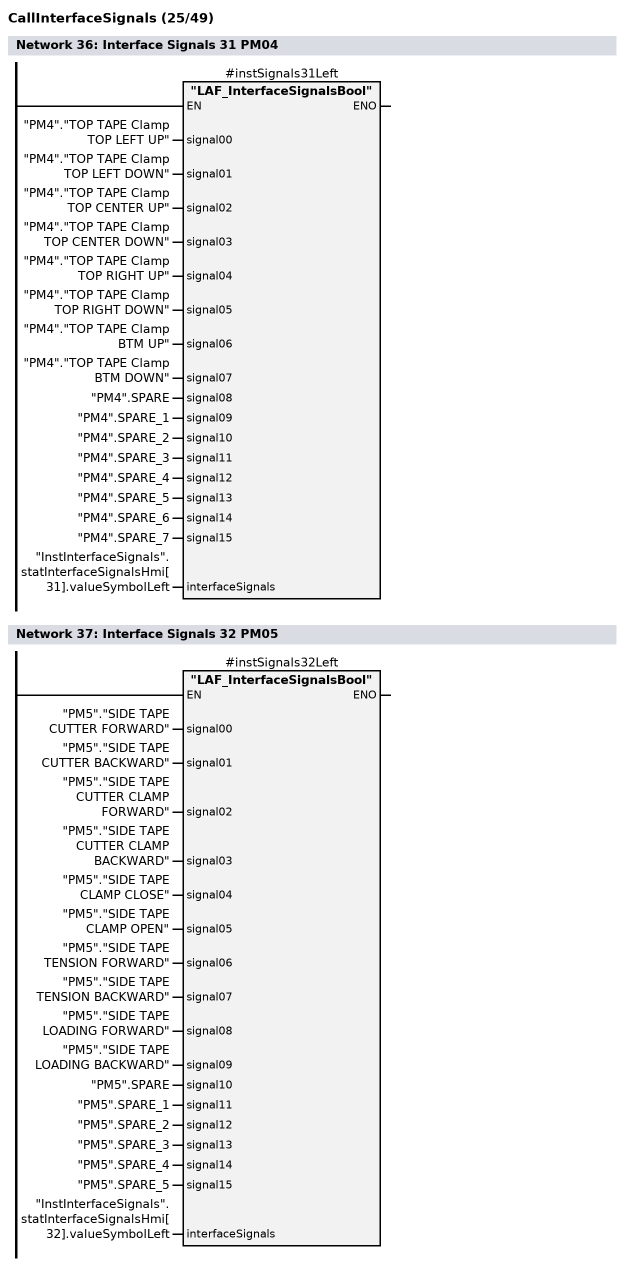
   RUNG wire#powerrail
      #instSignals31Left(signal00 := "PM4"."TOP TAPE Clamp TOP LEFT UP", signal01 := "PM4"."TOP TAPE Clamp TOP LEFT DOWN", signal02 := "PM4"."TOP TAPE Clamp TOP CENTER UP", signal03 := "PM4"."TOP TAPE Clamp TOP CENTER DOWN", signal04 := "PM4"."TOP TAPE Clamp TOP RIGHT UP", signal05 := "PM4"."TOP TAPE Clamp TOP RIGHT DOWN", signal06 := "PM4"."TOP TAPE Clamp BTM UP", signal07 := "PM4"."TOP TAPE Clamp BTM DOWN", signal08 := "PM4".SPARE, signal09 := "PM4".SPARE_1, signal10 := "PM4".SPARE_2, signal11 := "PM4".SPARE_3, signal12 := "PM4".SPARE_4, signal13 := "PM4".SPARE_5, signal14 := "PM4".SPARE_6, signal15 := "PM4".SPARE_7, interfaceSignals := "InstInterfaceSignals".statInterfaceSignalsHmi[31].valueSymbolLeft)
   END_RUNG
   // the same network as SCL:
   #instSignals31Left(signal00 := "PM4"."TOP TAPE Clamp TOP LEFT UP",   // "LAF_InterfaceSignalsBool"
                      signal01 := "PM4"."TOP TAPE Clamp TOP LEFT DOWN",
                      signal02 := "PM4"."TOP TAPE Clamp TOP CENTER UP",
                      signal03 := "PM4"."TOP TAPE Clamp TOP CENTER DOWN",
                      signal04 := "PM4"."TOP TAPE Clamp TOP RIGHT UP",
                      signal05 := "PM4"."TOP TAPE Clamp TOP RIGHT DOWN",
                      signal06 := "PM4"."TOP TAPE Clamp BTM UP",
                      signal07 := "PM4"."TOP TAPE Clamp BTM DOWN",
                      signal08 := "PM4".SPARE,
                      signal09 := "PM4".SPARE_1,
                      signal10 := "PM4".SPARE_2,
                      signal11 := "PM4".SPARE_3,
                      signal12 := "PM4".SPARE_4,
                      signal13 := "PM4".SPARE_5,
                      signal14 := "PM4".SPARE_6,
                      signal15 := "PM4".SPARE_7,
                      interfaceSignals := "InstInterfaceSignals".statInterfaceSignalsHmi[31].valueSymbolLeft);
END_REGION

REGION Network 37: Interface Signals 32 PM05
   RUNG wire#powerrail
      #instSignals32Left(signal00 := "PM5"."SIDE TAPE CUTTER FORWARD", signal01 := "PM5"."SIDE TAPE CUTTER BACKWARD", signal02 := "PM5"."SIDE TAPE CUTTER CLAMP FORWARD", signal03 := "PM5"."SIDE TAPE CUTTER CLAMP BACKWARD", signal04 := "PM5"."SIDE TAPE CLAMP CLOSE", signal05 := "PM5"."SIDE TAPE CLAMP OPEN", signal06 := "PM5"."SIDE TAPE TENSION FORWARD", signal07 := "PM5"."SIDE TAPE TENSION BACKWARD", signal08 := "PM5"."SIDE TAPE LOADING FORWARD", signal09 := "PM5"."SIDE TAPE LOADING BACKWARD", signal10 := "PM5".SPARE, signal11 := "PM5".SPARE_1, signal12 := "PM5".SPARE_2, signal13 := "PM5".SPARE_3, signal14 := "PM5".SPARE_4, signal15 := "PM5".SPARE_5, interfaceSignals := "InstInterfaceSignals".statInterfaceSignalsHmi[32].valueSymbolLeft)
   END_RUNG
   // the same network as SCL:
   #instSignals32Left(signal00 := "PM5"."SIDE TAPE CUTTER FORWARD",   // "LAF_InterfaceSignalsBool"
                      signal01 := "PM5"."SIDE TAPE CUTTER BACKWARD",
                      signal02 := "PM5"."SIDE TAPE CUTTER CLAMP FORWARD",
                      signal03 := "PM5"."SIDE TAPE CUTTER CLAMP BACKWARD",
                      signal04 := "PM5"."SIDE TAPE CLAMP CLOSE",
                      signal05 := "PM5"."SIDE TAPE CLAMP OPEN",
                      signal06 := "PM5"."SIDE TAPE TENSION FORWARD",
                      signal07 := "PM5"."SIDE TAPE TENSION BACKWARD",
                      signal08 := "PM5"."SIDE TAPE LOADING FORWARD",
                      signal09 := "PM5"."SIDE TAPE LOADING BACKWARD",
                      signal10 := "PM5".SPARE,
                      signal11 := "PM5".SPARE_1,
                      signal12 := "PM5".SPARE_2,
                      signal13 := "PM5".SPARE_3,
                      signal14 := "PM5".SPARE_4,
                      signal15 := "PM5".SPARE_5,
                      interfaceSignals := "InstInterfaceSignals".statInterfaceSignalsHmi[32].valueSymbolLeft);
END_REGION

REGION Network 38: Interface Signals 33 PM06
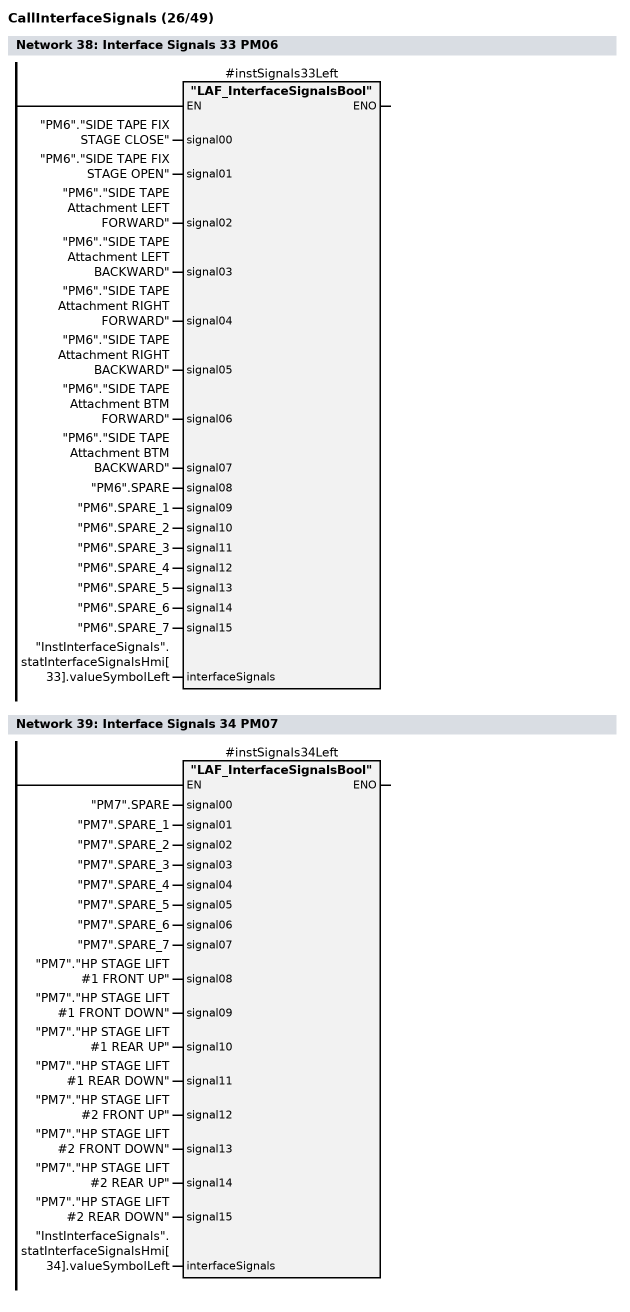
   RUNG wire#powerrail
      #instSignals33Left(signal00 := "PM6"."SIDE TAPE FIX STAGE CLOSE", signal01 := "PM6"."SIDE TAPE FIX STAGE OPEN", signal02 := "PM6"."SIDE TAPE Attachment LEFT FORWARD", signal03 := "PM6"."SIDE TAPE Attachment LEFT BACKWARD", signal04 := "PM6"."SIDE TAPE Attachment RIGHT FORWARD", signal05 := "PM6"."SIDE TAPE Attachment RIGHT BACKWARD", signal06 := "PM6"."SIDE TAPE Attachment BTM FORWARD", signal07 := "PM6"."SIDE TAPE Attachment BTM BACKWARD", signal08 := "PM6".SPARE, signal09 := "PM6".SPARE_1, signal10 := "PM6".SPARE_2, signal11 := "PM6".SPARE_3, signal12 := "PM6".SPARE_4, signal13 := "PM6".SPARE_5, signal14 := "PM6".SPARE_6, signal15 := "PM6".SPARE_7, interfaceSignals := "InstInterfaceSignals".statInterfaceSignalsHmi[33].valueSymbolLeft)
   END_RUNG
   // the same network as SCL:
   #instSignals33Left(signal00 := "PM6"."SIDE TAPE FIX STAGE CLOSE",   // "LAF_InterfaceSignalsBool"
                      signal01 := "PM6"."SIDE TAPE FIX STAGE OPEN",
                      signal02 := "PM6"."SIDE TAPE Attachment LEFT FORWARD",
                      signal03 := "PM6"."SIDE TAPE Attachment LEFT BACKWARD",
                      signal04 := "PM6"."SIDE TAPE Attachment RIGHT FORWARD",
                      signal05 := "PM6"."SIDE TAPE Attachment RIGHT BACKWARD",
                      signal06 := "PM6"."SIDE TAPE Attachment BTM FORWARD",
                      signal07 := "PM6"."SIDE TAPE Attachment BTM BACKWARD",
                      signal08 := "PM6".SPARE,
                      signal09 := "PM6".SPARE_1,
                      signal10 := "PM6".SPARE_2,
                      signal11 := "PM6".SPARE_3,
                      signal12 := "PM6".SPARE_4,
                      signal13 := "PM6".SPARE_5,
                      signal14 := "PM6".SPARE_6,
                      signal15 := "PM6".SPARE_7,
                      interfaceSignals := "InstInterfaceSignals".statInterfaceSignalsHmi[33].valueSymbolLeft);
END_REGION

REGION Network 39: Interface Signals 34 PM07
   RUNG wire#powerrail
      #instSignals34Left(signal00 := "PM7".SPARE, signal01 := "PM7".SPARE_1, signal02 := "PM7".SPARE_2, signal03 := "PM7".SPARE_3, signal04 := "PM7".SPARE_4, signal05 := "PM7".SPARE_5, signal06 := "PM7".SPARE_6, signal07 := "PM7".SPARE_7, signal08 := "PM7"."HP STAGE LIFT #1 FRONT UP", signal09 := "PM7"."HP STAGE LIFT #1 FRONT DOWN", signal10 := "PM7"."HP STAGE LIFT #1 REAR UP", signal11 := "PM7"."HP STAGE LIFT #1 REAR DOWN", signal12 := "PM7"."HP STAGE LIFT #2 FRONT UP", signal13 := "PM7"."HP STAGE LIFT #2 FRONT DOWN", signal14 := "PM7"."HP STAGE LIFT #2 REAR UP", signal15 := "PM7"."HP STAGE LIFT #2 REAR DOWN", interfaceSignals := "InstInterfaceSignals".statInterfaceSignalsHmi[34].valueSymbolLeft)
   END_RUNG
   // the same network as SCL:
   #instSignals34Left(signal00 := "PM7".SPARE,   // "LAF_InterfaceSignalsBool"
                      signal01 := "PM7".SPARE_1,
                      signal02 := "PM7".SPARE_2,
                      signal03 := "PM7".SPARE_3,
                      signal04 := "PM7".SPARE_4,
                      signal05 := "PM7".SPARE_5,
                      signal06 := "PM7".SPARE_6,
                      signal07 := "PM7".SPARE_7,
                      signal08 := "PM7"."HP STAGE LIFT #1 FRONT UP",
                      signal09 := "PM7"."HP STAGE LIFT #1 FRONT DOWN",
                      signal10 := "PM7"."HP STAGE LIFT #1 REAR UP",
                      signal11 := "PM7"."HP STAGE LIFT #1 REAR DOWN",
                      signal12 := "PM7"."HP STAGE LIFT #2 FRONT UP",
                      signal13 := "PM7"."HP STAGE LIFT #2 FRONT DOWN",
                      signal14 := "PM7"."HP STAGE LIFT #2 REAR UP",
                      signal15 := "PM7"."HP STAGE LIFT #2 REAR DOWN",
                      interfaceSignals := "InstInterfaceSignals".statInterfaceSignalsHmi[34].valueSymbolLeft);
END_REGION

REGION Network 40: Interface Signals 35 PM08
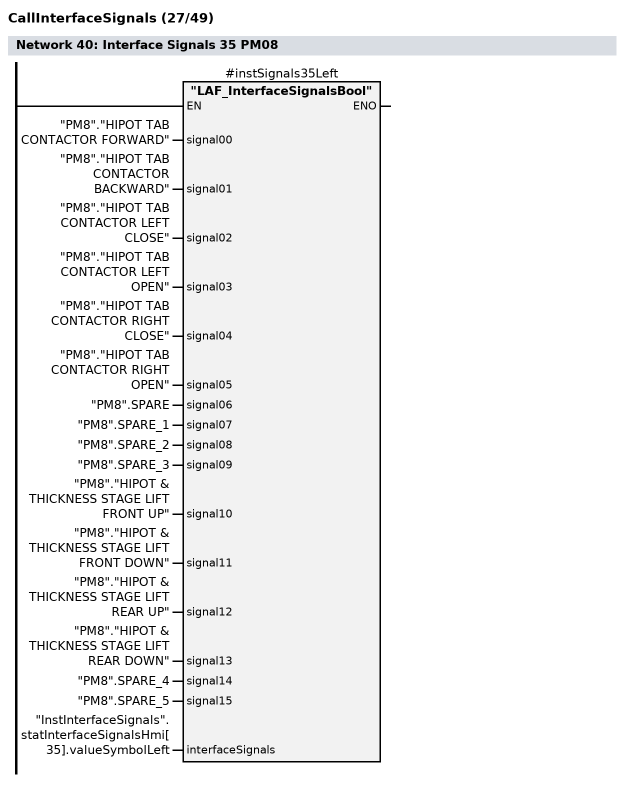
   RUNG wire#powerrail
      #instSignals35Left(signal00 := "PM8"."HIPOT TAB CONTACTOR FORWARD", signal01 := "PM8"."HIPOT TAB CONTACTOR BACKWARD", signal02 := "PM8"."HIPOT TAB CONTACTOR LEFT CLOSE", signal03 := "PM8"."HIPOT TAB CONTACTOR LEFT OPEN", signal04 := "PM8"."HIPOT TAB CONTACTOR RIGHT CLOSE", signal05 := "PM8"."HIPOT TAB CONTACTOR RIGHT OPEN", signal06 := "PM8".SPARE, signal07 := "PM8".SPARE_1, signal08 := "PM8".SPARE_2, signal09 := "PM8".SPARE_3, signal10 := "PM8"."HIPOT & THICKNESS STAGE LIFT FRONT UP", signal11 := "PM8"."HIPOT & THICKNESS STAGE LIFT FRONT DOWN", signal12 := "PM8"."HIPOT & THICKNESS STAGE LIFT REAR UP", signal13 := "PM8"."HIPOT & THICKNESS STAGE LIFT REAR DOWN", signal14 := "PM8".SPARE_4, signal15 := "PM8".SPARE_5, interfaceSignals := "InstInterfaceSignals".statInterfaceSignalsHmi[35].valueSymbolLeft)
   END_RUNG
   // the same network as SCL:
   #instSignals35Left(signal00 := "PM8"."HIPOT TAB CONTACTOR FORWARD",   // "LAF_InterfaceSignalsBool"
                      signal01 := "PM8"."HIPOT TAB CONTACTOR BACKWARD",
                      signal02 := "PM8"."HIPOT TAB CONTACTOR LEFT CLOSE",
                      signal03 := "PM8"."HIPOT TAB CONTACTOR LEFT OPEN",
                      signal04 := "PM8"."HIPOT TAB CONTACTOR RIGHT CLOSE",
                      signal05 := "PM8"."HIPOT TAB CONTACTOR RIGHT OPEN",
                      signal06 := "PM8".SPARE,
                      signal07 := "PM8".SPARE_1,
                      signal08 := "PM8".SPARE_2,
                      signal09 := "PM8".SPARE_3,
                      signal10 := "PM8"."HIPOT & THICKNESS STAGE LIFT FRONT UP",
                      signal11 := "PM8"."HIPOT & THICKNESS STAGE LIFT FRONT DOWN",
                      signal12 := "PM8"."HIPOT & THICKNESS STAGE LIFT REAR UP",
                      signal13 := "PM8"."HIPOT & THICKNESS STAGE LIFT REAR DOWN",
                      signal14 := "PM8".SPARE_4,
                      signal15 := "PM8".SPARE_5,
                      interfaceSignals := "InstInterfaceSignals".statInterfaceSignalsHmi[35].valueSymbolLeft);
END_REGION

REGION Network 41: Interface Signals 36 PM09
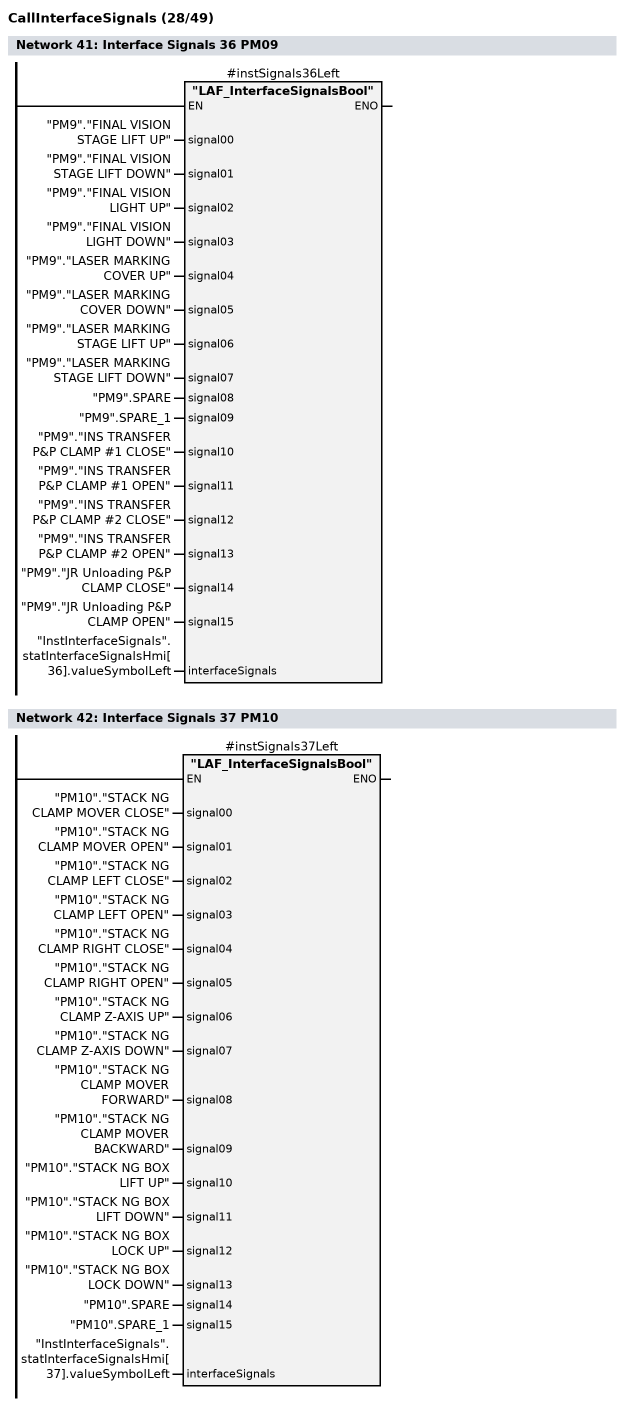
   RUNG wire#powerrail
      #instSignals36Left(signal00 := "PM9"."FINAL VISION STAGE LIFT UP", signal01 := "PM9"."FINAL VISION STAGE LIFT DOWN", signal02 := "PM9"."FINAL VISION LIGHT UP", signal03 := "PM9"."FINAL VISION LIGHT DOWN", signal04 := "PM9"."LASER MARKING COVER UP", signal05 := "PM9"."LASER MARKING COVER DOWN", signal06 := "PM9"."LASER MARKING STAGE LIFT UP", signal07 := "PM9"."LASER MARKING STAGE LIFT DOWN", signal08 := "PM9".SPARE, signal09 := "PM9".SPARE_1, signal10 := "PM9"."INS TRANSFER P&P CLAMP #1 CLOSE", signal11 := "PM9"."INS TRANSFER P&P CLAMP #1 OPEN", signal12 := "PM9"."INS TRANSFER P&P CLAMP #2 CLOSE", signal13 := "PM9"."INS TRANSFER P&P CLAMP #2 OPEN", signal14 := "PM9"."JR Unloading P&P CLAMP CLOSE", signal15 := "PM9"."JR Unloading P&P CLAMP OPEN", interfaceSignals := "InstInterfaceSignals".statInterfaceSignalsHmi[36].valueSymbolLeft)
   END_RUNG
   // the same network as SCL:
   #instSignals36Left(signal00 := "PM9"."FINAL VISION STAGE LIFT UP",   // "LAF_InterfaceSignalsBool"
                      signal01 := "PM9"."FINAL VISION STAGE LIFT DOWN",
                      signal02 := "PM9"."FINAL VISION LIGHT UP",
                      signal03 := "PM9"."FINAL VISION LIGHT DOWN",
                      signal04 := "PM9"."LASER MARKING COVER UP",
                      signal05 := "PM9"."LASER MARKING COVER DOWN",
                      signal06 := "PM9"."LASER MARKING STAGE LIFT UP",
                      signal07 := "PM9"."LASER MARKING STAGE LIFT DOWN",
                      signal08 := "PM9".SPARE,
                      signal09 := "PM9".SPARE_1,
                      signal10 := "PM9"."INS TRANSFER P&P CLAMP #1 CLOSE",
                      signal11 := "PM9"."INS TRANSFER P&P CLAMP #1 OPEN",
                      signal12 := "PM9"."INS TRANSFER P&P CLAMP #2 CLOSE",
                      signal13 := "PM9"."INS TRANSFER P&P CLAMP #2 OPEN",
                      signal14 := "PM9"."JR Unloading P&P CLAMP CLOSE",
                      signal15 := "PM9"."JR Unloading P&P CLAMP OPEN",
                      interfaceSignals := "InstInterfaceSignals".statInterfaceSignalsHmi[36].valueSymbolLeft);
END_REGION

REGION Network 42: Interface Signals 37 PM10
   RUNG wire#powerrail
      #instSignals37Left(signal00 := "PM10"."STACK NG CLAMP MOVER CLOSE", signal01 := "PM10"."STACK NG CLAMP MOVER OPEN", signal02 := "PM10"."STACK NG CLAMP LEFT CLOSE", signal03 := "PM10"."STACK NG CLAMP LEFT OPEN", signal04 := "PM10"."STACK NG CLAMP RIGHT CLOSE", signal05 := "PM10"."STACK NG CLAMP RIGHT OPEN", signal06 := "PM10"."STACK NG CLAMP Z-AXIS UP", signal07 := "PM10"."STACK NG CLAMP Z-AXIS DOWN", signal08 := "PM10"."STACK NG CLAMP MOVER FORWARD", signal09 := "PM10"."STACK NG CLAMP MOVER BACKWARD", signal10 := "PM10"."STACK NG BOX LIFT UP", signal11 := "PM10"."STACK NG BOX LIFT DOWN", signal12 := "PM10"."STACK NG BOX LOCK UP", signal13 := "PM10"."STACK NG BOX LOCK DOWN", signal14 := "PM10".SPARE, signal15 := "PM10".SPARE_1, interfaceSignals := "InstInterfaceSignals".statInterfaceSignalsHmi[37].valueSymbolLeft)
   END_RUNG
   // the same network as SCL:
   #instSignals37Left(signal00 := "PM10"."STACK NG CLAMP MOVER CLOSE",   // "LAF_InterfaceSignalsBool"
                      signal01 := "PM10"."STACK NG CLAMP MOVER OPEN",
                      signal02 := "PM10"."STACK NG CLAMP LEFT CLOSE",
                      signal03 := "PM10"."STACK NG CLAMP LEFT OPEN",
                      signal04 := "PM10"."STACK NG CLAMP RIGHT CLOSE",
                      signal05 := "PM10"."STACK NG CLAMP RIGHT OPEN",
                      signal06 := "PM10"."STACK NG CLAMP Z-AXIS UP",
                      signal07 := "PM10"."STACK NG CLAMP Z-AXIS DOWN",
                      signal08 := "PM10"."STACK NG CLAMP MOVER FORWARD",
                      signal09 := "PM10"."STACK NG CLAMP MOVER BACKWARD",
                      signal10 := "PM10"."STACK NG BOX LIFT UP",
                      signal11 := "PM10"."STACK NG BOX LIFT DOWN",
                      signal12 := "PM10"."STACK NG BOX LOCK UP",
                      signal13 := "PM10"."STACK NG BOX LOCK DOWN",
                      signal14 := "PM10".SPARE,
                      signal15 := "PM10".SPARE_1,
                      interfaceSignals := "InstInterfaceSignals".statInterfaceSignalsHmi[37].valueSymbolLeft);
END_REGION

REGION Network 43: Interface Signals 38 SBK01
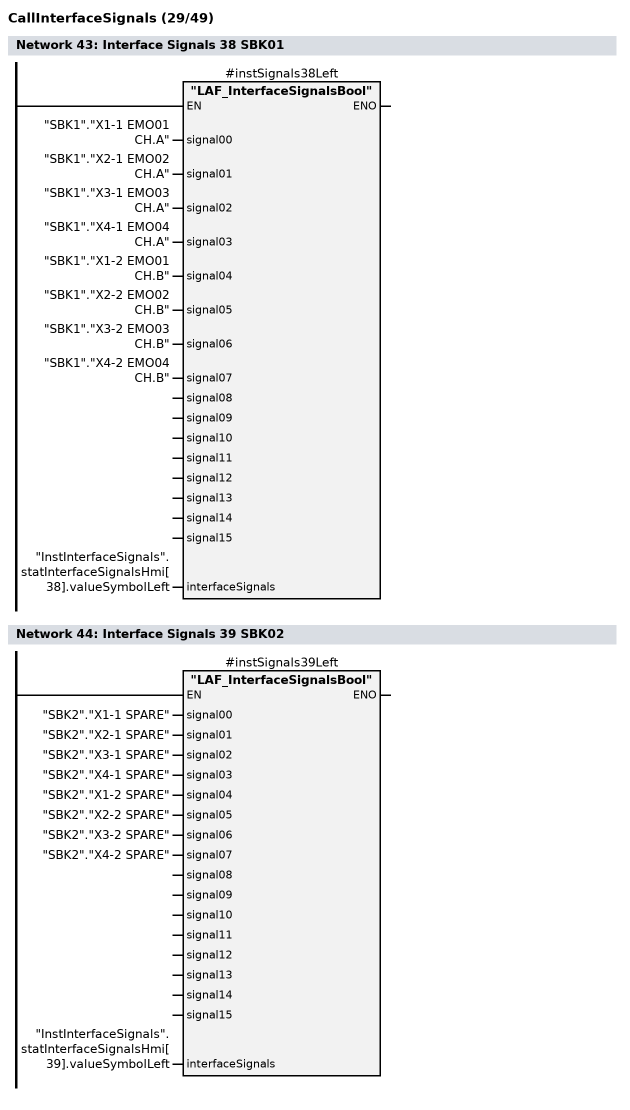
   RUNG wire#powerrail
      #instSignals38Left(signal00 := "SBK1"."X1-1 EMO01 CH.A", signal01 := "SBK1"."X2-1 EMO02 CH.A", signal02 := "SBK1"."X3-1 EMO03 CH.A", signal03 := "SBK1"."X4-1 EMO04 CH.A", signal04 := "SBK1"."X1-2 EMO01 CH.B", signal05 := "SBK1"."X2-2 EMO02 CH.B", signal06 := "SBK1"."X3-2 EMO03 CH.B", signal07 := "SBK1"."X4-2 EMO04 CH.B", signal08 :=, signal09 :=, signal10 :=, signal11 :=, signal12 :=, signal13 :=, signal14 :=, signal15 :=, interfaceSignals := "InstInterfaceSignals".statInterfaceSignalsHmi[38].valueSymbolLeft)
   END_RUNG
   // the same network as SCL:
   #instSignals38Left(signal00 := "SBK1"."X1-1 EMO01 CH.A",   // "LAF_InterfaceSignalsBool"
                      signal01 := "SBK1"."X2-1 EMO02 CH.A",
                      signal02 := "SBK1"."X3-1 EMO03 CH.A",
                      signal03 := "SBK1"."X4-1 EMO04 CH.A",
                      signal04 := "SBK1"."X1-2 EMO01 CH.B",
                      signal05 := "SBK1"."X2-2 EMO02 CH.B",
                      signal06 := "SBK1"."X3-2 EMO03 CH.B",
                      signal07 := "SBK1"."X4-2 EMO04 CH.B",
                      interfaceSignals := "InstInterfaceSignals".statInterfaceSignalsHmi[38].valueSymbolLeft);
END_REGION

REGION Network 44: Interface Signals 39 SBK02
   RUNG wire#powerrail
      #instSignals39Left(signal00 := "SBK2"."X1-1 SPARE", signal01 := "SBK2"."X2-1 SPARE", signal02 := "SBK2"."X3-1 SPARE", signal03 := "SBK2"."X4-1 SPARE", signal04 := "SBK2"."X1-2 SPARE", signal05 := "SBK2"."X2-2 SPARE", signal06 := "SBK2"."X3-2 SPARE", signal07 := "SBK2"."X4-2 SPARE", signal08 :=, signal09 :=, signal10 :=, signal11 :=, signal12 :=, signal13 :=, signal14 :=, signal15 :=, interfaceSignals := "InstInterfaceSignals".statInterfaceSignalsHmi[39].valueSymbolLeft)
   END_RUNG
   // the same network as SCL:
   #instSignals39Left(signal00 := "SBK2"."X1-1 SPARE",   // "LAF_InterfaceSignalsBool"
                      signal01 := "SBK2"."X2-1 SPARE",
                      signal02 := "SBK2"."X3-1 SPARE",
                      signal03 := "SBK2"."X4-1 SPARE",
                      signal04 := "SBK2"."X1-2 SPARE",
                      signal05 := "SBK2"."X2-2 SPARE",
                      signal06 := "SBK2"."X3-2 SPARE",
                      signal07 := "SBK2"."X4-2 SPARE",
                      interfaceSignals := "InstInterfaceSignals".statInterfaceSignalsHmi[39].valueSymbolLeft);
END_REGION

REGION Network 45: Interface Signals 40 SBK03
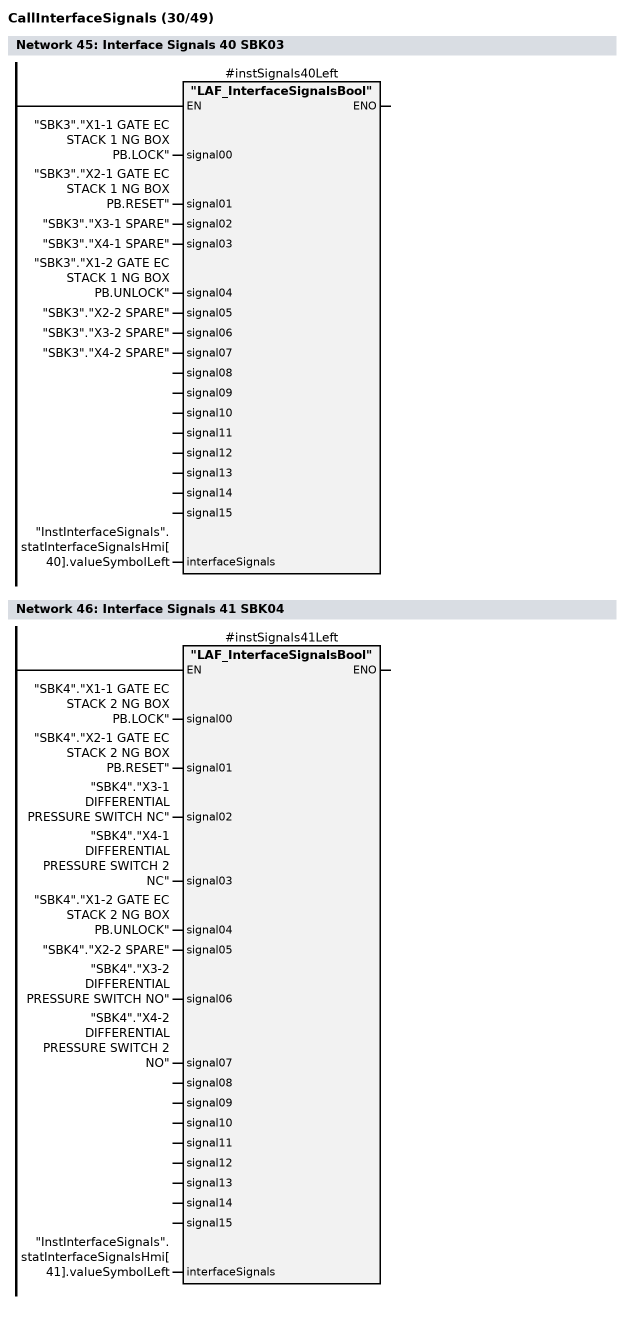
   RUNG wire#powerrail
      #instSignals40Left(signal00 := "SBK3"."X1-1 GATE EC STACK 1 NG BOX PB.LOCK", signal01 := "SBK3"."X2-1 GATE EC STACK 1 NG BOX PB.RESET", signal02 := "SBK3"."X3-1 SPARE", signal03 := "SBK3"."X4-1 SPARE", signal04 := "SBK3"."X1-2 GATE EC STACK 1 NG BOX PB.UNLOCK", signal05 := "SBK3"."X2-2 SPARE", signal06 := "SBK3"."X3-2 SPARE", signal07 := "SBK3"."X4-2 SPARE", signal08 :=, signal09 :=, signal10 :=, signal11 :=, signal12 :=, signal13 :=, signal14 :=, signal15 :=, interfaceSignals := "InstInterfaceSignals".statInterfaceSignalsHmi[40].valueSymbolLeft)
   END_RUNG
   // the same network as SCL:
   #instSignals40Left(signal00 := "SBK3"."X1-1 GATE EC STACK 1 NG BOX PB.LOCK",   // "LAF_InterfaceSignalsBool"
                      signal01 := "SBK3"."X2-1 GATE EC STACK 1 NG BOX PB.RESET",
                      signal02 := "SBK3"."X3-1 SPARE",
                      signal03 := "SBK3"."X4-1 SPARE",
                      signal04 := "SBK3"."X1-2 GATE EC STACK 1 NG BOX PB.UNLOCK",
                      signal05 := "SBK3"."X2-2 SPARE",
                      signal06 := "SBK3"."X3-2 SPARE",
                      signal07 := "SBK3"."X4-2 SPARE",
                      interfaceSignals := "InstInterfaceSignals".statInterfaceSignalsHmi[40].valueSymbolLeft);
END_REGION

REGION Network 46: Interface Signals 41 SBK04
   RUNG wire#powerrail
      #instSignals41Left(signal00 := "SBK4"."X1-1 GATE EC STACK 2 NG BOX PB.LOCK", signal01 := "SBK4"."X2-1 GATE EC STACK 2 NG BOX PB.RESET", signal02 := "SBK4"."X3-1 DIFFERENTIAL PRESSURE SWITCH NC", signal03 := "SBK4"."X4-1 DIFFERENTIAL PRESSURE SWITCH 2 NC", signal04 := "SBK4"."X1-2 GATE EC STACK 2 NG BOX PB.UNLOCK", signal05 := "SBK4"."X2-2 SPARE", signal06 := "SBK4"."X3-2 DIFFERENTIAL PRESSURE SWITCH NO", signal07 := "SBK4"."X4-2 DIFFERENTIAL PRESSURE SWITCH 2 NO", signal08 :=, signal09 :=, signal10 :=, signal11 :=, signal12 :=, signal13 :=, signal14 :=, signal15 :=, interfaceSignals := "InstInterfaceSignals".statInterfaceSignalsHmi[41].valueSymbolLeft)
   END_RUNG
   // the same network as SCL:
   #instSignals41Left(signal00 := "SBK4"."X1-1 GATE EC STACK 2 NG BOX PB.LOCK",   // "LAF_InterfaceSignalsBool"
                      signal01 := "SBK4"."X2-1 GATE EC STACK 2 NG BOX PB.RESET",
                      signal02 := "SBK4"."X3-1 DIFFERENTIAL PRESSURE SWITCH NC",
                      signal03 := "SBK4"."X4-1 DIFFERENTIAL PRESSURE SWITCH 2 NC",
                      signal04 := "SBK4"."X1-2 GATE EC STACK 2 NG BOX PB.UNLOCK",
                      signal05 := "SBK4"."X2-2 SPARE",
                      signal06 := "SBK4"."X3-2 DIFFERENTIAL PRESSURE SWITCH NO",
                      signal07 := "SBK4"."X4-2 DIFFERENTIAL PRESSURE SWITCH 2 NO",
                      interfaceSignals := "InstInterfaceSignals".statInterfaceSignalsHmi[41].valueSymbolLeft);
END_REGION

REGION Network 47: Interface Signals 42 SBK05
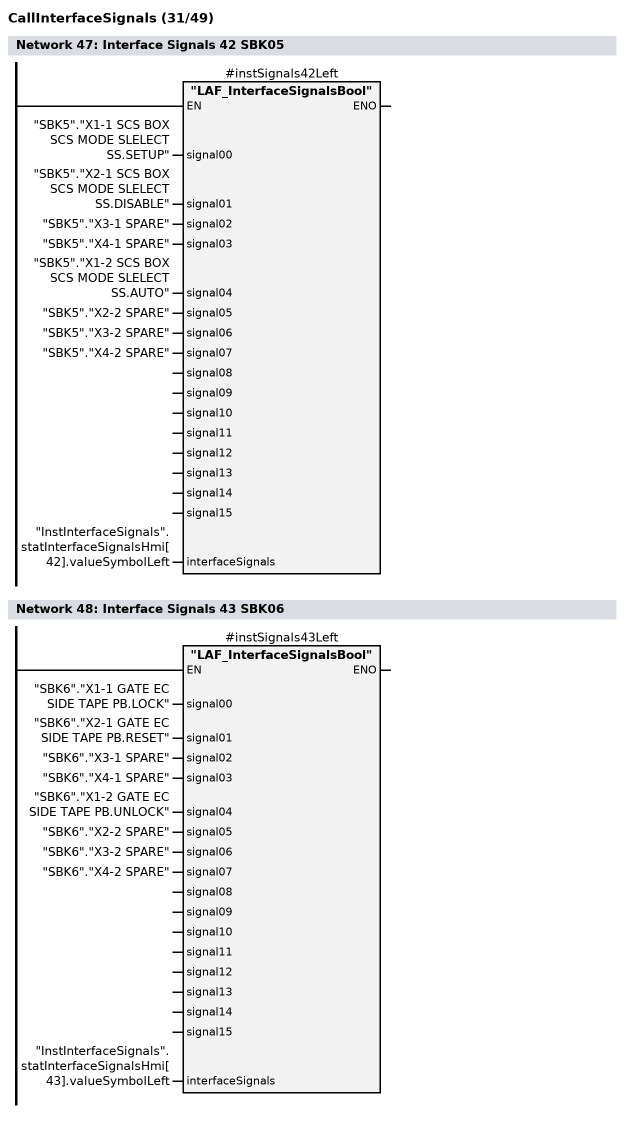
   RUNG wire#powerrail
      #instSignals42Left(signal00 := "SBK5"."X1-1 SCS BOX SCS MODE SLELECT SS.SETUP", signal01 := "SBK5"."X2-1 SCS BOX SCS MODE SLELECT SS.DISABLE", signal02 := "SBK5"."X3-1 SPARE", signal03 := "SBK5"."X4-1 SPARE", signal04 := "SBK5"."X1-2 SCS BOX SCS MODE SLELECT SS.AUTO", signal05 := "SBK5"."X2-2 SPARE", signal06 := "SBK5"."X3-2 SPARE", signal07 := "SBK5"."X4-2 SPARE", signal08 :=, signal09 :=, signal10 :=, signal11 :=, signal12 :=, signal13 :=, signal14 :=, signal15 :=, interfaceSignals := "InstInterfaceSignals".statInterfaceSignalsHmi[42].valueSymbolLeft)
   END_RUNG
   // the same network as SCL:
   #instSignals42Left(signal00 := "SBK5"."X1-1 SCS BOX SCS MODE SLELECT SS.SETUP",   // "LAF_InterfaceSignalsBool"
                      signal01 := "SBK5"."X2-1 SCS BOX SCS MODE SLELECT SS.DISABLE",
                      signal02 := "SBK5"."X3-1 SPARE",
                      signal03 := "SBK5"."X4-1 SPARE",
                      signal04 := "SBK5"."X1-2 SCS BOX SCS MODE SLELECT SS.AUTO",
                      signal05 := "SBK5"."X2-2 SPARE",
                      signal06 := "SBK5"."X3-2 SPARE",
                      signal07 := "SBK5"."X4-2 SPARE",
                      interfaceSignals := "InstInterfaceSignals".statInterfaceSignalsHmi[42].valueSymbolLeft);
END_REGION

REGION Network 48: Interface Signals 43 SBK06
   RUNG wire#powerrail
      #instSignals43Left(signal00 := "SBK6"."X1-1 GATE EC SIDE TAPE PB.LOCK", signal01 := "SBK6"."X2-1 GATE EC SIDE TAPE PB.RESET", signal02 := "SBK6"."X3-1 SPARE", signal03 := "SBK6"."X4-1 SPARE", signal04 := "SBK6"."X1-2 GATE EC SIDE TAPE PB.UNLOCK", signal05 := "SBK6"."X2-2 SPARE", signal06 := "SBK6"."X3-2 SPARE", signal07 := "SBK6"."X4-2 SPARE", signal08 :=, signal09 :=, signal10 :=, signal11 :=, signal12 :=, signal13 :=, signal14 :=, signal15 :=, interfaceSignals := "InstInterfaceSignals".statInterfaceSignalsHmi[43].valueSymbolLeft)
   END_RUNG
   // the same network as SCL:
   #instSignals43Left(signal00 := "SBK6"."X1-1 GATE EC SIDE TAPE PB.LOCK",   // "LAF_InterfaceSignalsBool"
                      signal01 := "SBK6"."X2-1 GATE EC SIDE TAPE PB.RESET",
                      signal02 := "SBK6"."X3-1 SPARE",
                      signal03 := "SBK6"."X4-1 SPARE",
                      signal04 := "SBK6"."X1-2 GATE EC SIDE TAPE PB.UNLOCK",
                      signal05 := "SBK6"."X2-2 SPARE",
                      signal06 := "SBK6"."X3-2 SPARE",
                      signal07 := "SBK6"."X4-2 SPARE",
                      interfaceSignals := "InstInterfaceSignals".statInterfaceSignalsHmi[43].valueSymbolLeft);
END_REGION

REGION Network 49: Interface Signals 44 SBK07
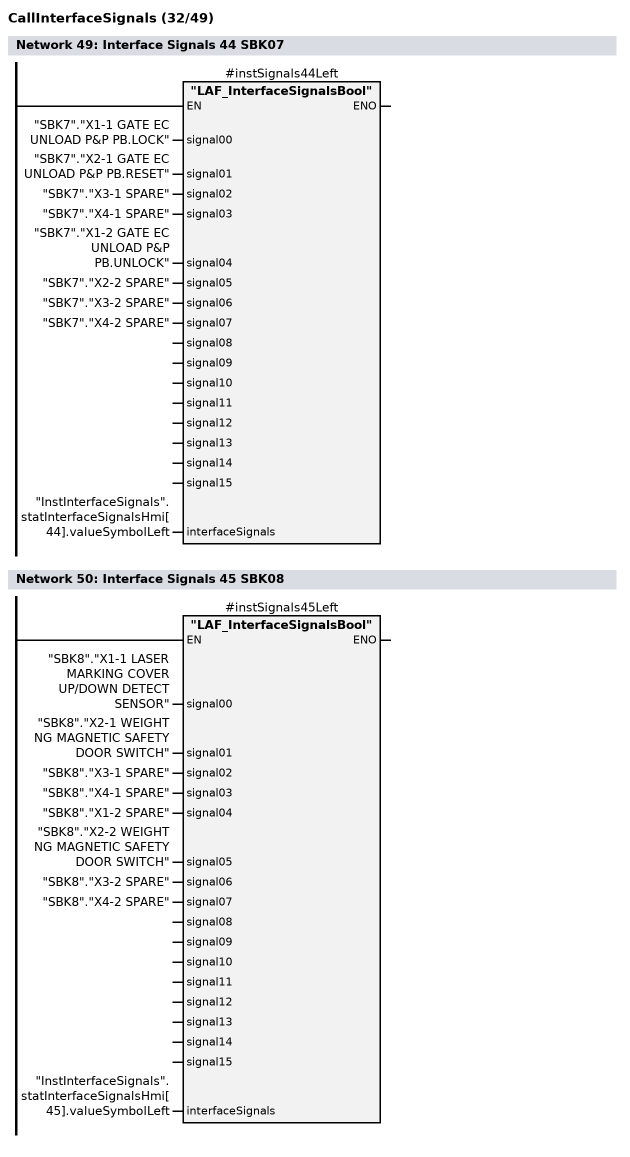
   RUNG wire#powerrail
      #instSignals44Left(signal00 := "SBK7"."X1-1 GATE EC UNLOAD P&P PB.LOCK", signal01 := "SBK7"."X2-1 GATE EC UNLOAD P&P PB.RESET", signal02 := "SBK7"."X3-1 SPARE", signal03 := "SBK7"."X4-1 SPARE", signal04 := "SBK7"."X1-2 GATE EC UNLOAD P&P PB.UNLOCK", signal05 := "SBK7"."X2-2 SPARE", signal06 := "SBK7"."X3-2 SPARE", signal07 := "SBK7"."X4-2 SPARE", signal08 :=, signal09 :=, signal10 :=, signal11 :=, signal12 :=, signal13 :=, signal14 :=, signal15 :=, interfaceSignals := "InstInterfaceSignals".statInterfaceSignalsHmi[44].valueSymbolLeft)
   END_RUNG
   // the same network as SCL:
   #instSignals44Left(signal00 := "SBK7"."X1-1 GATE EC UNLOAD P&P PB.LOCK",   // "LAF_InterfaceSignalsBool"
                      signal01 := "SBK7"."X2-1 GATE EC UNLOAD P&P PB.RESET",
                      signal02 := "SBK7"."X3-1 SPARE",
                      signal03 := "SBK7"."X4-1 SPARE",
                      signal04 := "SBK7"."X1-2 GATE EC UNLOAD P&P PB.UNLOCK",
                      signal05 := "SBK7"."X2-2 SPARE",
                      signal06 := "SBK7"."X3-2 SPARE",
                      signal07 := "SBK7"."X4-2 SPARE",
                      interfaceSignals := "InstInterfaceSignals".statInterfaceSignalsHmi[44].valueSymbolLeft);
END_REGION

REGION Network 50: Interface Signals 45 SBK08
   RUNG wire#powerrail
      #instSignals45Left(signal00 := "SBK8"."X1-1 LASER MARKING COVER UP/DOWN DETECT SENSOR", signal01 := "SBK8"."X2-1 WEIGHT NG MAGNETIC SAFETY DOOR SWITCH", signal02 := "SBK8"."X3-1 SPARE", signal03 := "SBK8"."X4-1 SPARE", signal04 := "SBK8"."X1-2 SPARE", signal05 := "SBK8"."X2-2 WEIGHT NG MAGNETIC SAFETY DOOR SWITCH", signal06 := "SBK8"."X3-2 SPARE", signal07 := "SBK8"."X4-2 SPARE", signal08 :=, signal09 :=, signal10 :=, signal11 :=, signal12 :=, signal13 :=, signal14 :=, signal15 :=, interfaceSignals := "InstInterfaceSignals".statInterfaceSignalsHmi[45].valueSymbolLeft)
   END_RUNG
   // the same network as SCL:
   #instSignals45Left(signal00 := "SBK8"."X1-1 LASER MARKING COVER UP/DOWN DETECT SENSOR",   // "LAF_InterfaceSignalsBool"
                      signal01 := "SBK8"."X2-1 WEIGHT NG MAGNETIC SAFETY DOOR SWITCH",
                      signal02 := "SBK8"."X3-1 SPARE",
                      signal03 := "SBK8"."X4-1 SPARE",
                      signal04 := "SBK8"."X1-2 SPARE",
                      signal05 := "SBK8"."X2-2 WEIGHT NG MAGNETIC SAFETY DOOR SWITCH",
                      signal06 := "SBK8"."X3-2 SPARE",
                      signal07 := "SBK8"."X4-2 SPARE",
                      interfaceSignals := "InstInterfaceSignals".statInterfaceSignalsHmi[45].valueSymbolLeft);
END_REGION

REGION Network 51: Interface Signals 46 SBK09
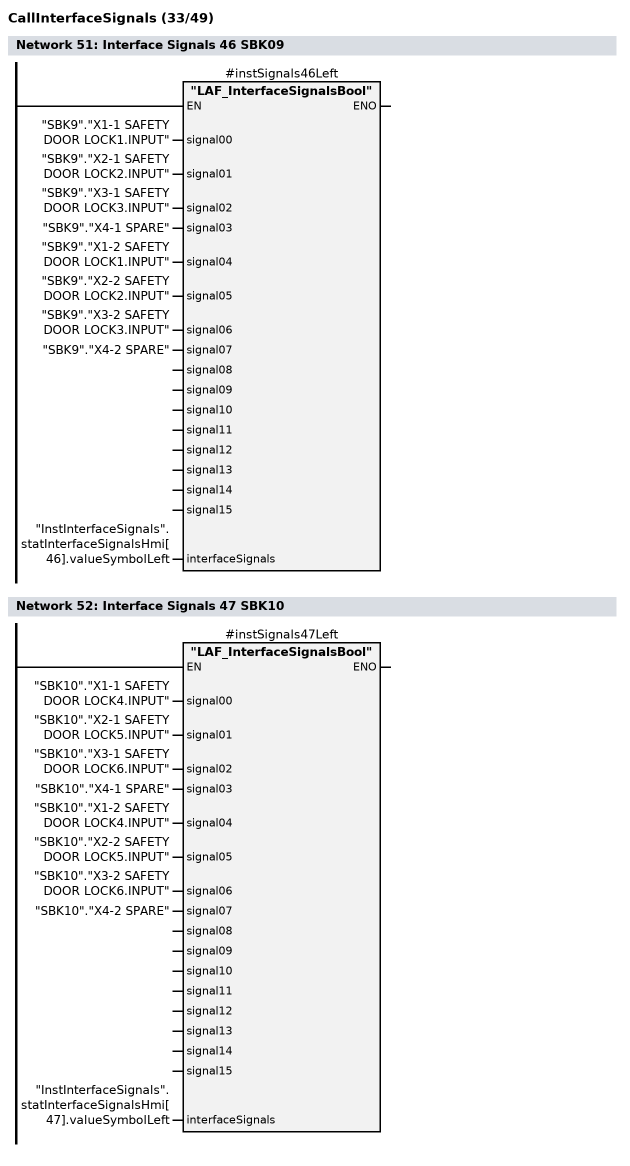
   RUNG wire#powerrail
      #instSignals46Left(signal00 := "SBK9"."X1-1 SAFETY DOOR LOCK1.INPUT", signal01 := "SBK9"."X2-1 SAFETY DOOR LOCK2.INPUT", signal02 := "SBK9"."X3-1 SAFETY DOOR LOCK3.INPUT", signal03 := "SBK9"."X4-1 SPARE", signal04 := "SBK9"."X1-2 SAFETY DOOR LOCK1.INPUT", signal05 := "SBK9"."X2-2 SAFETY DOOR LOCK2.INPUT", signal06 := "SBK9"."X3-2 SAFETY DOOR LOCK3.INPUT", signal07 := "SBK9"."X4-2 SPARE", signal08 :=, signal09 :=, signal10 :=, signal11 :=, signal12 :=, signal13 :=, signal14 :=, signal15 :=, interfaceSignals := "InstInterfaceSignals".statInterfaceSignalsHmi[46].valueSymbolLeft)
   END_RUNG
   // the same network as SCL:
   #instSignals46Left(signal00 := "SBK9"."X1-1 SAFETY DOOR LOCK1.INPUT",   // "LAF_InterfaceSignalsBool"
                      signal01 := "SBK9"."X2-1 SAFETY DOOR LOCK2.INPUT",
                      signal02 := "SBK9"."X3-1 SAFETY DOOR LOCK3.INPUT",
                      signal03 := "SBK9"."X4-1 SPARE",
                      signal04 := "SBK9"."X1-2 SAFETY DOOR LOCK1.INPUT",
                      signal05 := "SBK9"."X2-2 SAFETY DOOR LOCK2.INPUT",
                      signal06 := "SBK9"."X3-2 SAFETY DOOR LOCK3.INPUT",
                      signal07 := "SBK9"."X4-2 SPARE",
                      interfaceSignals := "InstInterfaceSignals".statInterfaceSignalsHmi[46].valueSymbolLeft);
END_REGION

REGION Network 52: Interface Signals 47 SBK10
   RUNG wire#powerrail
      #instSignals47Left(signal00 := "SBK10"."X1-1 SAFETY DOOR LOCK4.INPUT", signal01 := "SBK10"."X2-1 SAFETY DOOR LOCK5.INPUT", signal02 := "SBK10"."X3-1 SAFETY DOOR LOCK6.INPUT", signal03 := "SBK10"."X4-1 SPARE", signal04 := "SBK10"."X1-2 SAFETY DOOR LOCK4.INPUT", signal05 := "SBK10"."X2-2 SAFETY DOOR LOCK5.INPUT", signal06 := "SBK10"."X3-2 SAFETY DOOR LOCK6.INPUT", signal07 := "SBK10"."X4-2 SPARE", signal08 :=, signal09 :=, signal10 :=, signal11 :=, signal12 :=, signal13 :=, signal14 :=, signal15 :=, interfaceSignals := "InstInterfaceSignals".statInterfaceSignalsHmi[47].valueSymbolLeft)
   END_RUNG
   // the same network as SCL:
   #instSignals47Left(signal00 := "SBK10"."X1-1 SAFETY DOOR LOCK4.INPUT",   // "LAF_InterfaceSignalsBool"
                      signal01 := "SBK10"."X2-1 SAFETY DOOR LOCK5.INPUT",
                      signal02 := "SBK10"."X3-1 SAFETY DOOR LOCK6.INPUT",
                      signal03 := "SBK10"."X4-1 SPARE",
                      signal04 := "SBK10"."X1-2 SAFETY DOOR LOCK4.INPUT",
                      signal05 := "SBK10"."X2-2 SAFETY DOOR LOCK5.INPUT",
                      signal06 := "SBK10"."X3-2 SAFETY DOOR LOCK6.INPUT",
                      signal07 := "SBK10"."X4-2 SPARE",
                      interfaceSignals := "InstInterfaceSignals".statInterfaceSignalsHmi[47].valueSymbolLeft);
END_REGION

REGION Network 53: Interface Signals 48 SBK11
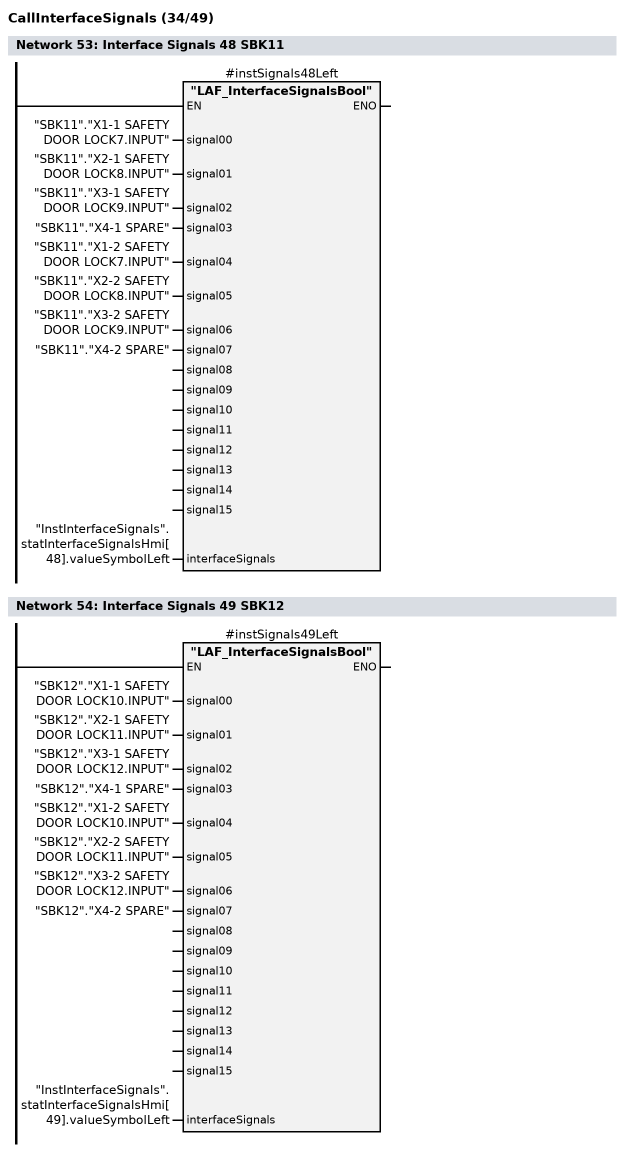
   RUNG wire#powerrail
      #instSignals48Left(signal00 := "SBK11"."X1-1 SAFETY DOOR LOCK7.INPUT", signal01 := "SBK11"."X2-1 SAFETY DOOR LOCK8.INPUT", signal02 := "SBK11"."X3-1 SAFETY DOOR LOCK9.INPUT", signal03 := "SBK11"."X4-1 SPARE", signal04 := "SBK11"."X1-2 SAFETY DOOR LOCK7.INPUT", signal05 := "SBK11"."X2-2 SAFETY DOOR LOCK8.INPUT", signal06 := "SBK11"."X3-2 SAFETY DOOR LOCK9.INPUT", signal07 := "SBK11"."X4-2 SPARE", signal08 :=, signal09 :=, signal10 :=, signal11 :=, signal12 :=, signal13 :=, signal14 :=, signal15 :=, interfaceSignals := "InstInterfaceSignals".statInterfaceSignalsHmi[48].valueSymbolLeft)
   END_RUNG
   // the same network as SCL:
   #instSignals48Left(signal00 := "SBK11"."X1-1 SAFETY DOOR LOCK7.INPUT",   // "LAF_InterfaceSignalsBool"
                      signal01 := "SBK11"."X2-1 SAFETY DOOR LOCK8.INPUT",
                      signal02 := "SBK11"."X3-1 SAFETY DOOR LOCK9.INPUT",
                      signal03 := "SBK11"."X4-1 SPARE",
                      signal04 := "SBK11"."X1-2 SAFETY DOOR LOCK7.INPUT",
                      signal05 := "SBK11"."X2-2 SAFETY DOOR LOCK8.INPUT",
                      signal06 := "SBK11"."X3-2 SAFETY DOOR LOCK9.INPUT",
                      signal07 := "SBK11"."X4-2 SPARE",
                      interfaceSignals := "InstInterfaceSignals".statInterfaceSignalsHmi[48].valueSymbolLeft);
END_REGION

REGION Network 54: Interface Signals 49 SBK12
   RUNG wire#powerrail
      #instSignals49Left(signal00 := "SBK12"."X1-1 SAFETY DOOR LOCK10.INPUT", signal01 := "SBK12"."X2-1 SAFETY DOOR LOCK11.INPUT", signal02 := "SBK12"."X3-1 SAFETY DOOR LOCK12.INPUT", signal03 := "SBK12"."X4-1 SPARE", signal04 := "SBK12"."X1-2 SAFETY DOOR LOCK10.INPUT", signal05 := "SBK12"."X2-2 SAFETY DOOR LOCK11.INPUT", signal06 := "SBK12"."X3-2 SAFETY DOOR LOCK12.INPUT", signal07 := "SBK12"."X4-2 SPARE", signal08 :=, signal09 :=, signal10 :=, signal11 :=, signal12 :=, signal13 :=, signal14 :=, signal15 :=, interfaceSignals := "InstInterfaceSignals".statInterfaceSignalsHmi[49].valueSymbolLeft)
   END_RUNG
   // the same network as SCL:
   #instSignals49Left(signal00 := "SBK12"."X1-1 SAFETY DOOR LOCK10.INPUT",   // "LAF_InterfaceSignalsBool"
                      signal01 := "SBK12"."X2-1 SAFETY DOOR LOCK11.INPUT",
                      signal02 := "SBK12"."X3-1 SAFETY DOOR LOCK12.INPUT",
                      signal03 := "SBK12"."X4-1 SPARE",
                      signal04 := "SBK12"."X1-2 SAFETY DOOR LOCK10.INPUT",
                      signal05 := "SBK12"."X2-2 SAFETY DOOR LOCK11.INPUT",
                      signal06 := "SBK12"."X3-2 SAFETY DOOR LOCK12.INPUT",
                      signal07 := "SBK12"."X4-2 SPARE",
                      interfaceSignals := "InstInterfaceSignals".statInterfaceSignalsHmi[49].valueSymbolLeft);
END_REGION

REGION Network 55: Interface Signals 50 SBK13
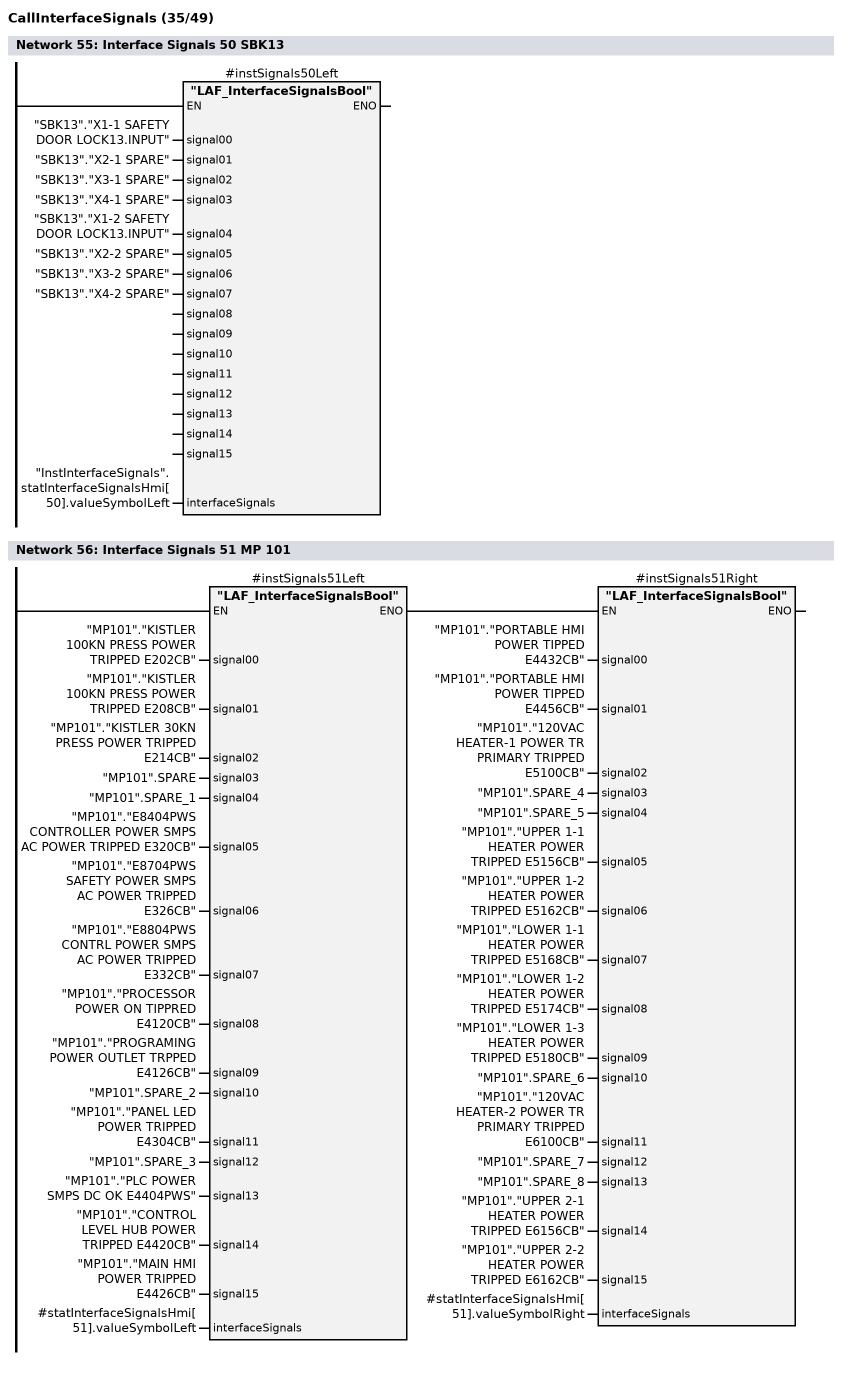
   RUNG wire#powerrail
      #instSignals50Left(signal00 := "SBK13"."X1-1 SAFETY DOOR LOCK13.INPUT", signal01 := "SBK13"."X2-1 SPARE", signal02 := "SBK13"."X3-1 SPARE", signal03 := "SBK13"."X4-1 SPARE", signal04 := "SBK13"."X1-2 SAFETY DOOR LOCK13.INPUT", signal05 := "SBK13"."X2-2 SPARE", signal06 := "SBK13"."X3-2 SPARE", signal07 := "SBK13"."X4-2 SPARE", signal08 :=, signal09 :=, signal10 :=, signal11 :=, signal12 :=, signal13 :=, signal14 :=, signal15 :=, interfaceSignals := "InstInterfaceSignals".statInterfaceSignalsHmi[50].valueSymbolLeft)
   END_RUNG
   // the same network as SCL:
   #instSignals50Left(signal00 := "SBK13"."X1-1 SAFETY DOOR LOCK13.INPUT",   // "LAF_InterfaceSignalsBool"
                      signal01 := "SBK13"."X2-1 SPARE",
                      signal02 := "SBK13"."X3-1 SPARE",
                      signal03 := "SBK13"."X4-1 SPARE",
                      signal04 := "SBK13"."X1-2 SAFETY DOOR LOCK13.INPUT",
                      signal05 := "SBK13"."X2-2 SPARE",
                      signal06 := "SBK13"."X3-2 SPARE",
                      signal07 := "SBK13"."X4-2 SPARE",
                      interfaceSignals := "InstInterfaceSignals".statInterfaceSignalsHmi[50].valueSymbolLeft);
END_REGION

REGION Network 56: Interface Signals 51 MP 101
   RUNG wire#powerrail
      #instSignals51Left(signal00 := "MP101"."KISTLER 100KN PRESS POWER TRIPPED E202CB", signal01 := "MP101"."KISTLER 100KN PRESS POWER TRIPPED E208CB", signal02 := "MP101"."KISTLER 30KN PRESS POWER TRIPPED E214CB", signal03 := "MP101".SPARE, signal04 := "MP101".SPARE_1, signal05 := "MP101"."E8404PWS CONTROLLER POWER SMPS AC POWER TRIPPED E320CB", signal06 := "MP101"."E8704PWS SAFETY POWER SMPS AC POWER TRIPPED E326CB", signal07 := "MP101"."E8804PWS CONTRL POWER SMPS AC POWER TRIPPED E332CB", signal08 := "MP101"."PROCESSOR POWER ON TIPPRED E4120CB", signal09 := "MP101"."PROGRAMING POWER OUTLET TRPPED E4126CB", signal10 := "MP101".SPARE_2, signal11 := "MP101"."PANEL LED POWER TRIPPED E4304CB", signal12 := "MP101".SPARE_3, signal13 := "MP101"."PLC POWER SMPS DC OK E4404PWS", signal14 := "MP101"."CONTROL LEVEL HUB POWER TRIPPED E4420CB", signal15 := "MP101"."MAIN HMI POWER TRIPPED E4426CB", interfaceSignals := #statInterfaceSignalsHmi[51].valueSymbolLeft)
      #instSignals51Right(signal00 := "MP101"."PORTABLE HMI POWER TIPPED E4432CB", signal01 := "MP101"."PORTABLE HMI POWER TIPPED E4456CB", signal02 := "MP101"."120VAC HEATER-1 POWER TR PRIMARY TRIPPED E5100CB", signal03 := "MP101".SPARE_4, signal04 := "MP101".SPARE_5, signal05 := "MP101"."UPPER 1-1 HEATER POWER TRIPPED E5156CB", signal06 := "MP101"."UPPER 1-2 HEATER POWER TRIPPED E5162CB", signal07 := "MP101"."LOWER 1-1 HEATER POWER TRIPPED E5168CB", signal08 := "MP101"."LOWER 1-2 HEATER POWER TRIPPED E5174CB", signal09 := "MP101"."LOWER 1-3 HEATER POWER TRIPPED E5180CB", signal10 := "MP101".SPARE_6, signal11 := "MP101"."120VAC HEATER-2 POWER TR PRIMARY TRIPPED E6100CB", signal12 := "MP101".SPARE_7, signal13 := "MP101".SPARE_8, signal14 := "MP101"."UPPER 2-1 HEATER POWER TRIPPED E6156CB", signal15 := "MP101"."UPPER 2-2 HEATER POWER TRIPPED E6162CB", interfaceSignals := #statInterfaceSignalsHmi[51].valueSymbolRight)
   END_RUNG
   // the same network as SCL:
   #instSignals51Left(signal00 := "MP101"."KISTLER 100KN PRESS POWER TRIPPED E202CB",   // "LAF_InterfaceSignalsBool"
                      signal01 := "MP101"."KISTLER 100KN PRESS POWER TRIPPED E208CB",
                      signal02 := "MP101"."KISTLER 30KN PRESS POWER TRIPPED E214CB",
                      signal03 := "MP101".SPARE,
                      signal04 := "MP101".SPARE_1,
                      signal05 := "MP101"."E8404PWS CONTROLLER POWER SMPS AC POWER TRIPPED E320CB",
                      signal06 := "MP101"."E8704PWS SAFETY POWER SMPS AC POWER TRIPPED E326CB",
                      signal07 := "MP101"."E8804PWS CONTRL POWER SMPS AC POWER TRIPPED E332CB",
                      signal08 := "MP101"."PROCESSOR POWER ON TIPPRED E4120CB",
                      signal09 := "MP101"."PROGRAMING POWER OUTLET TRPPED E4126CB",
                      signal10 := "MP101".SPARE_2,
                      signal11 := "MP101"."PANEL LED POWER TRIPPED E4304CB",
                      signal12 := "MP101".SPARE_3,
                      signal13 := "MP101"."PLC POWER SMPS DC OK E4404PWS",
                      signal14 := "MP101"."CONTROL LEVEL HUB POWER TRIPPED E4420CB",
                      signal15 := "MP101"."MAIN HMI POWER TRIPPED E4426CB",
                      interfaceSignals := #statInterfaceSignalsHmi[51].valueSymbolLeft,
                      ENO => #_w1);
   IF #_w1 THEN
       #instSignals51Right(signal00 := "MP101"."PORTABLE HMI POWER TIPPED E4432CB",   // "LAF_InterfaceSignalsBool"
                           signal01 := "MP101"."PORTABLE HMI POWER TIPPED E4456CB",
                           signal02 := "MP101"."120VAC HEATER-1 POWER TR PRIMARY TRIPPED E5100CB",
                           signal03 := "MP101".SPARE_4,
                           signal04 := "MP101".SPARE_5,
                           signal05 := "MP101"."UPPER 1-1 HEATER POWER TRIPPED E5156CB",
                           signal06 := "MP101"."UPPER 1-2 HEATER POWER TRIPPED E5162CB",
                           signal07 := "MP101"."LOWER 1-1 HEATER POWER TRIPPED E5168CB",
                           signal08 := "MP101"."LOWER 1-2 HEATER POWER TRIPPED E5174CB",
                           signal09 := "MP101"."LOWER 1-3 HEATER POWER TRIPPED E5180CB",
                           signal10 := "MP101".SPARE_6,
                           signal11 := "MP101"."120VAC HEATER-2 POWER TR PRIMARY TRIPPED E6100CB",
                           signal12 := "MP101".SPARE_7,
                           signal13 := "MP101".SPARE_8,
                           signal14 := "MP101"."UPPER 2-1 HEATER POWER TRIPPED E6156CB",
                           signal15 := "MP101"."UPPER 2-2 HEATER POWER TRIPPED E6162CB",
                           interfaceSignals := #statInterfaceSignalsHmi[51].valueSymbolRight);
   END_IF;
END_REGION

REGION Network 57: Interface Signals 52 MP 102
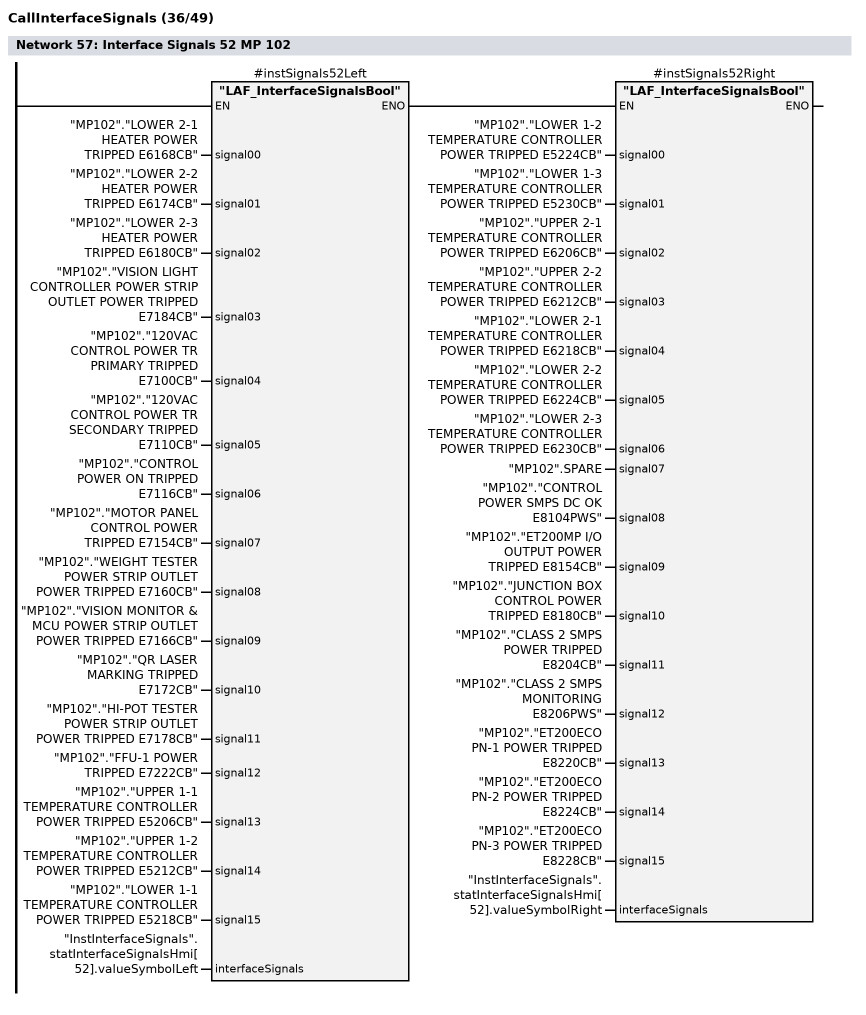
   RUNG wire#powerrail
      #instSignals52Left(signal00 := "MP102"."LOWER 2-1 HEATER POWER TRIPPED E6168CB", signal01 := "MP102"."LOWER 2-2 HEATER POWER TRIPPED E6174CB", signal02 := "MP102"."LOWER 2-3 HEATER POWER TRIPPED E6180CB", signal03 := "MP102"."VISION LIGHT CONTROLLER POWER STRIP OUTLET POWER TRIPPED E7184CB", signal04 := "MP102"."120VAC CONTROL POWER TR PRIMARY TRIPPED E7100CB", signal05 := "MP102"."120VAC CONTROL POWER TR SECONDARY TRIPPED E7110CB", signal06 := "MP102"."CONTROL POWER ON TRIPPED E7116CB", signal07 := "MP102"."MOTOR PANEL CONTROL POWER TRIPPED E7154CB", signal08 := "MP102"."WEIGHT TESTER POWER STRIP OUTLET POWER TRIPPED E7160CB", signal09 := "MP102"."VISION MONITOR & MCU POWER STRIP OUTLET POWER TRIPPED E7166CB", signal10 := "MP102"."QR LASER MARKING TRIPPED E7172CB", signal11 := "MP102"."HI-POT TESTER POWER STRIP OUTLET POWER TRIPPED E7178CB", signal12 := "MP102"."FFU-1 POWER TRIPPED E7222CB", signal13 := "MP102"."UPPER 1-1 TEMPERATURE CONTROLLER POWER TRIPPED E5206CB", signal14 := "MP102"."UPPER 1-2 TEMPERATURE CONTROLLER POWER TRIPPED E5212CB", signal15 := "MP102"."LOWER 1-1 TEMPERATURE CONTROLLER POWER TRIPPED E5218CB", interfaceSignals := "InstInterfaceSignals".statInterfaceSignalsHmi[52].valueSymbolLeft)
      #instSignals52Right(signal00 := "MP102"."LOWER 1-2 TEMPERATURE CONTROLLER POWER TRIPPED E5224CB", signal01 := "MP102"."LOWER 1-3 TEMPERATURE CONTROLLER POWER TRIPPED E5230CB", signal02 := "MP102"."UPPER 2-1 TEMPERATURE CONTROLLER POWER TRIPPED E6206CB", signal03 := "MP102"."UPPER 2-2 TEMPERATURE CONTROLLER POWER TRIPPED E6212CB", signal04 := "MP102"."LOWER 2-1 TEMPERATURE CONTROLLER POWER TRIPPED E6218CB", signal05 := "MP102"."LOWER 2-2 TEMPERATURE CONTROLLER POWER TRIPPED E6224CB", signal06 := "MP102"."LOWER 2-3 TEMPERATURE CONTROLLER POWER TRIPPED E6230CB", signal07 := "MP102".SPARE, signal08 := "MP102"."CONTROL POWER SMPS DC OK E8104PWS", signal09 := "MP102"."ET200MP I/O OUTPUT POWER TRIPPED E8154CB", signal10 := "MP102"."JUNCTION BOX CONTROL POWER TRIPPED E8180CB", signal11 := "MP102"."CLASS 2 SMPS POWER TRIPPED E8204CB", signal12 := "MP102"."CLASS 2 SMPS MONITORING E8206PWS", signal13 := "MP102"."ET200ECO PN-1 POWER TRIPPED E8220CB", signal14 := "MP102"."ET200ECO PN-2 POWER TRIPPED E8224CB", signal15 := "MP102"."ET200ECO PN-3 POWER TRIPPED E8228CB", interfaceSignals := "InstInterfaceSignals".statInterfaceSignalsHmi[52].valueSymbolRight)
   END_RUNG
   // the same network as SCL:
   #instSignals52Left(signal00 := "MP102"."LOWER 2-1 HEATER POWER TRIPPED E6168CB",   // "LAF_InterfaceSignalsBool"
                      signal01 := "MP102"."LOWER 2-2 HEATER POWER TRIPPED E6174CB",
                      signal02 := "MP102"."LOWER 2-3 HEATER POWER TRIPPED E6180CB",
                      signal03 := "MP102"."VISION LIGHT CONTROLLER POWER STRIP OUTLET POWER TRIPPED E7184CB",
                      signal04 := "MP102"."120VAC CONTROL POWER TR PRIMARY TRIPPED E7100CB",
                      signal05 := "MP102"."120VAC CONTROL POWER TR SECONDARY TRIPPED E7110CB",
                      signal06 := "MP102"."CONTROL POWER ON TRIPPED E7116CB",
                      signal07 := "MP102"."MOTOR PANEL CONTROL POWER TRIPPED E7154CB",
                      signal08 := "MP102"."WEIGHT TESTER POWER STRIP OUTLET POWER TRIPPED E7160CB",
                      signal09 := "MP102"."VISION MONITOR & MCU POWER STRIP OUTLET POWER TRIPPED E7166CB",
                      signal10 := "MP102"."QR LASER MARKING TRIPPED E7172CB",
                      signal11 := "MP102"."HI-POT TESTER POWER STRIP OUTLET POWER TRIPPED E7178CB",
                      signal12 := "MP102"."FFU-1 POWER TRIPPED E7222CB",
                      signal13 := "MP102"."UPPER 1-1 TEMPERATURE CONTROLLER POWER TRIPPED E5206CB",
                      signal14 := "MP102"."UPPER 1-2 TEMPERATURE CONTROLLER POWER TRIPPED E5212CB",
                      signal15 := "MP102"."LOWER 1-1 TEMPERATURE CONTROLLER POWER TRIPPED E5218CB",
                      interfaceSignals := "InstInterfaceSignals".statInterfaceSignalsHmi[52].valueSymbolLeft,
                      ENO => #_w1);
   IF #_w1 THEN
       #instSignals52Right(signal00 := "MP102"."LOWER 1-2 TEMPERATURE CONTROLLER POWER TRIPPED E5224CB",   // "LAF_InterfaceSignalsBool"
                           signal01 := "MP102"."LOWER 1-3 TEMPERATURE CONTROLLER POWER TRIPPED E5230CB",
                           signal02 := "MP102"."UPPER 2-1 TEMPERATURE CONTROLLER POWER TRIPPED E6206CB",
                           signal03 := "MP102"."UPPER 2-2 TEMPERATURE CONTROLLER POWER TRIPPED E6212CB",
                           signal04 := "MP102"."LOWER 2-1 TEMPERATURE CONTROLLER POWER TRIPPED E6218CB",
                           signal05 := "MP102"."LOWER 2-2 TEMPERATURE CONTROLLER POWER TRIPPED E6224CB",
                           signal06 := "MP102"."LOWER 2-3 TEMPERATURE CONTROLLER POWER TRIPPED E6230CB",
                           signal07 := "MP102".SPARE,
                           signal08 := "MP102"."CONTROL POWER SMPS DC OK E8104PWS",
                           signal09 := "MP102"."ET200MP I/O OUTPUT POWER TRIPPED E8154CB",
                           signal10 := "MP102"."JUNCTION BOX CONTROL POWER TRIPPED E8180CB",
                           signal11 := "MP102"."CLASS 2 SMPS POWER TRIPPED E8204CB",
                           signal12 := "MP102"."CLASS 2 SMPS MONITORING E8206PWS",
                           signal13 := "MP102"."ET200ECO PN-1 POWER TRIPPED E8220CB",
                           signal14 := "MP102"."ET200ECO PN-2 POWER TRIPPED E8224CB",
                           signal15 := "MP102"."ET200ECO PN-3 POWER TRIPPED E8228CB",
                           interfaceSignals := "InstInterfaceSignals".statInterfaceSignalsHmi[52].valueSymbolRight);
   END_IF;
END_REGION

REGION Network 58: Interface Signals 53 MP 103
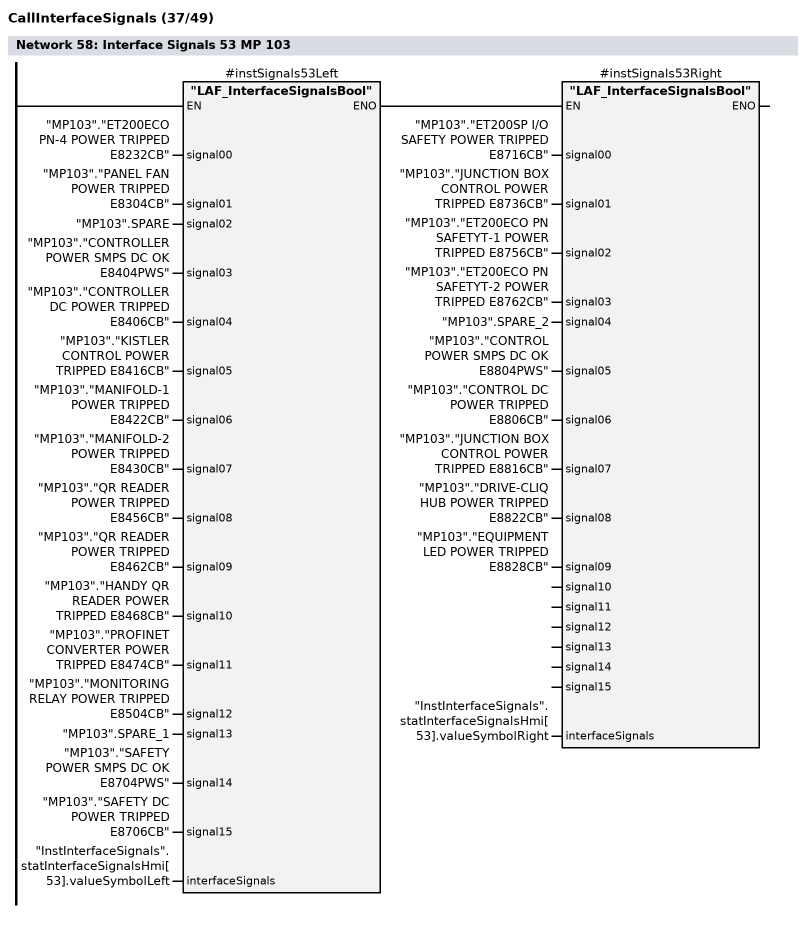
   RUNG wire#powerrail
      #instSignals53Left(signal00 := "MP103"."ET200ECO PN-4 POWER TRIPPED E8232CB", signal01 := "MP103"."PANEL FAN POWER TRIPPED E8304CB", signal02 := "MP103".SPARE, signal03 := "MP103"."CONTROLLER POWER SMPS DC OK E8404PWS", signal04 := "MP103"."CONTROLLER DC POWER TRIPPED E8406CB", signal05 := "MP103"."KISTLER CONTROL POWER TRIPPED E8416CB", signal06 := "MP103"."MANIFOLD-1 POWER TRIPPED E8422CB", signal07 := "MP103"."MANIFOLD-2 POWER TRIPPED E8430CB", signal08 := "MP103"."QR READER POWER TRIPPED E8456CB", signal09 := "MP103"."QR READER POWER TRIPPED E8462CB", signal10 := "MP103"."HANDY QR READER POWER TRIPPED E8468CB", signal11 := "MP103"."PROFINET CONVERTER POWER TRIPPED E8474CB", signal12 := "MP103"."MONITORING RELAY POWER TRIPPED E8504CB", signal13 := "MP103".SPARE_1, signal14 := "MP103"."SAFETY POWER SMPS DC OK E8704PWS", signal15 := "MP103"."SAFETY DC POWER TRIPPED E8706CB", interfaceSignals := "InstInterfaceSignals".statInterfaceSignalsHmi[53].valueSymbolLeft)
      #instSignals53Right(signal00 := "MP103"."ET200SP I/O SAFETY POWER TRIPPED E8716CB", signal01 := "MP103"."JUNCTION BOX CONTROL POWER TRIPPED E8736CB", signal02 := "MP103"."ET200ECO PN SAFETYT-1 POWER TRIPPED E8756CB", signal03 := "MP103"."ET200ECO PN SAFETYT-2 POWER TRIPPED E8762CB", signal04 := "MP103".SPARE_2, signal05 := "MP103"."CONTROL POWER SMPS DC OK E8804PWS", signal06 := "MP103"."CONTROL DC POWER TRIPPED E8806CB", signal07 := "MP103"."JUNCTION BOX CONTROL POWER TRIPPED E8816CB", signal08 := "MP103"."DRIVE-CLIQ HUB POWER TRIPPED E8822CB", signal09 := "MP103"."EQUIPMENT LED POWER TRIPPED E8828CB", signal10 :=, signal11 :=, signal12 :=, signal13 :=, signal14 :=, signal15 :=, interfaceSignals := "InstInterfaceSignals".statInterfaceSignalsHmi[53].valueSymbolRight)
   END_RUNG
   // the same network as SCL:
   #instSignals53Left(signal00 := "MP103"."ET200ECO PN-4 POWER TRIPPED E8232CB",   // "LAF_InterfaceSignalsBool"
                      signal01 := "MP103"."PANEL FAN POWER TRIPPED E8304CB",
                      signal02 := "MP103".SPARE,
                      signal03 := "MP103"."CONTROLLER POWER SMPS DC OK E8404PWS",
                      signal04 := "MP103"."CONTROLLER DC POWER TRIPPED E8406CB",
                      signal05 := "MP103"."KISTLER CONTROL POWER TRIPPED E8416CB",
                      signal06 := "MP103"."MANIFOLD-1 POWER TRIPPED E8422CB",
                      signal07 := "MP103"."MANIFOLD-2 POWER TRIPPED E8430CB",
                      signal08 := "MP103"."QR READER POWER TRIPPED E8456CB",
                      signal09 := "MP103"."QR READER POWER TRIPPED E8462CB",
                      signal10 := "MP103"."HANDY QR READER POWER TRIPPED E8468CB",
                      signal11 := "MP103"."PROFINET CONVERTER POWER TRIPPED E8474CB",
                      signal12 := "MP103"."MONITORING RELAY POWER TRIPPED E8504CB",
                      signal13 := "MP103".SPARE_1,
                      signal14 := "MP103"."SAFETY POWER SMPS DC OK E8704PWS",
                      signal15 := "MP103"."SAFETY DC POWER TRIPPED E8706CB",
                      interfaceSignals := "InstInterfaceSignals".statInterfaceSignalsHmi[53].valueSymbolLeft,
                      ENO => #_w1);
   IF #_w1 THEN
       #instSignals53Right(signal00 := "MP103"."ET200SP I/O SAFETY POWER TRIPPED E8716CB",   // "LAF_InterfaceSignalsBool"
                           signal01 := "MP103"."JUNCTION BOX CONTROL POWER TRIPPED E8736CB",
                           signal02 := "MP103"."ET200ECO PN SAFETYT-1 POWER TRIPPED E8756CB",
                           signal03 := "MP103"."ET200ECO PN SAFETYT-2 POWER TRIPPED E8762CB",
                           signal04 := "MP103".SPARE_2,
                           signal05 := "MP103"."CONTROL POWER SMPS DC OK E8804PWS",
                           signal06 := "MP103"."CONTROL DC POWER TRIPPED E8806CB",
                           signal07 := "MP103"."JUNCTION BOX CONTROL POWER TRIPPED E8816CB",
                           signal08 := "MP103"."DRIVE-CLIQ HUB POWER TRIPPED E8822CB",
                           signal09 := "MP103"."EQUIPMENT LED POWER TRIPPED E8828CB",
                           interfaceSignals := "InstInterfaceSignals".statInterfaceSignalsHmi[53].valueSymbolRight);
   END_IF;
END_REGION

REGION Network 59: Interface Signals 54 MP 104
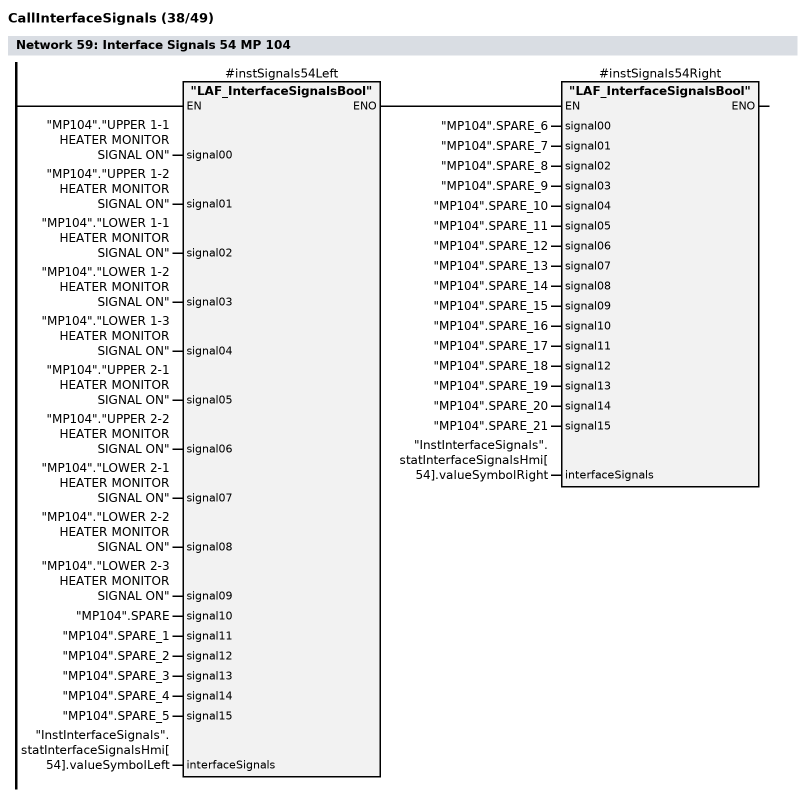
   RUNG wire#powerrail
      #instSignals54Left(signal00 := "MP104"."UPPER 1-1 HEATER MONITOR SIGNAL ON", signal01 := "MP104"."UPPER 1-2 HEATER MONITOR SIGNAL ON", signal02 := "MP104"."LOWER 1-1 HEATER MONITOR SIGNAL ON", signal03 := "MP104"."LOWER 1-2 HEATER MONITOR SIGNAL ON", signal04 := "MP104"."LOWER 1-3 HEATER MONITOR SIGNAL ON", signal05 := "MP104"."UPPER 2-1 HEATER MONITOR SIGNAL ON", signal06 := "MP104"."UPPER 2-2 HEATER MONITOR SIGNAL ON", signal07 := "MP104"."LOWER 2-1 HEATER MONITOR SIGNAL ON", signal08 := "MP104"."LOWER 2-2 HEATER MONITOR SIGNAL ON", signal09 := "MP104"."LOWER 2-3 HEATER MONITOR SIGNAL ON", signal10 := "MP104".SPARE, signal11 := "MP104".SPARE_1, signal12 := "MP104".SPARE_2, signal13 := "MP104".SPARE_3, signal14 := "MP104".SPARE_4, signal15 := "MP104".SPARE_5, interfaceSignals := "InstInterfaceSignals".statInterfaceSignalsHmi[54].valueSymbolLeft)
      #instSignals54Right(signal00 := "MP104".SPARE_6, signal01 := "MP104".SPARE_7, signal02 := "MP104".SPARE_8, signal03 := "MP104".SPARE_9, signal04 := "MP104".SPARE_10, signal05 := "MP104".SPARE_11, signal06 := "MP104".SPARE_12, signal07 := "MP104".SPARE_13, signal08 := "MP104".SPARE_14, signal09 := "MP104".SPARE_15, signal10 := "MP104".SPARE_16, signal11 := "MP104".SPARE_17, signal12 := "MP104".SPARE_18, signal13 := "MP104".SPARE_19, signal14 := "MP104".SPARE_20, signal15 := "MP104".SPARE_21, interfaceSignals := "InstInterfaceSignals".statInterfaceSignalsHmi[54].valueSymbolRight)
   END_RUNG
   // the same network as SCL:
   #instSignals54Left(signal00 := "MP104"."UPPER 1-1 HEATER MONITOR SIGNAL ON",   // "LAF_InterfaceSignalsBool"
                      signal01 := "MP104"."UPPER 1-2 HEATER MONITOR SIGNAL ON",
                      signal02 := "MP104"."LOWER 1-1 HEATER MONITOR SIGNAL ON",
                      signal03 := "MP104"."LOWER 1-2 HEATER MONITOR SIGNAL ON",
                      signal04 := "MP104"."LOWER 1-3 HEATER MONITOR SIGNAL ON",
                      signal05 := "MP104"."UPPER 2-1 HEATER MONITOR SIGNAL ON",
                      signal06 := "MP104"."UPPER 2-2 HEATER MONITOR SIGNAL ON",
                      signal07 := "MP104"."LOWER 2-1 HEATER MONITOR SIGNAL ON",
                      signal08 := "MP104"."LOWER 2-2 HEATER MONITOR SIGNAL ON",
                      signal09 := "MP104"."LOWER 2-3 HEATER MONITOR SIGNAL ON",
                      signal10 := "MP104".SPARE,
                      signal11 := "MP104".SPARE_1,
                      signal12 := "MP104".SPARE_2,
                      signal13 := "MP104".SPARE_3,
                      signal14 := "MP104".SPARE_4,
                      signal15 := "MP104".SPARE_5,
                      interfaceSignals := "InstInterfaceSignals".statInterfaceSignalsHmi[54].valueSymbolLeft,
                      ENO => #_w1);
   IF #_w1 THEN
       #instSignals54Right(signal00 := "MP104".SPARE_6,   // "LAF_InterfaceSignalsBool"
                           signal01 := "MP104".SPARE_7,
                           signal02 := "MP104".SPARE_8,
                           signal03 := "MP104".SPARE_9,
                           signal04 := "MP104".SPARE_10,
                           signal05 := "MP104".SPARE_11,
                           signal06 := "MP104".SPARE_12,
                           signal07 := "MP104".SPARE_13,
                           signal08 := "MP104".SPARE_14,
                           signal09 := "MP104".SPARE_15,
                           signal10 := "MP104".SPARE_16,
                           signal11 := "MP104".SPARE_17,
                           signal12 := "MP104".SPARE_18,
                           signal13 := "MP104".SPARE_19,
                           signal14 := "MP104".SPARE_20,
                           signal15 := "MP104".SPARE_21,
                           interfaceSignals := "InstInterfaceSignals".statInterfaceSignalsHmi[54].valueSymbolRight);
   END_IF;
END_REGION

REGION Network 60: Interface Signals 55 MP 105
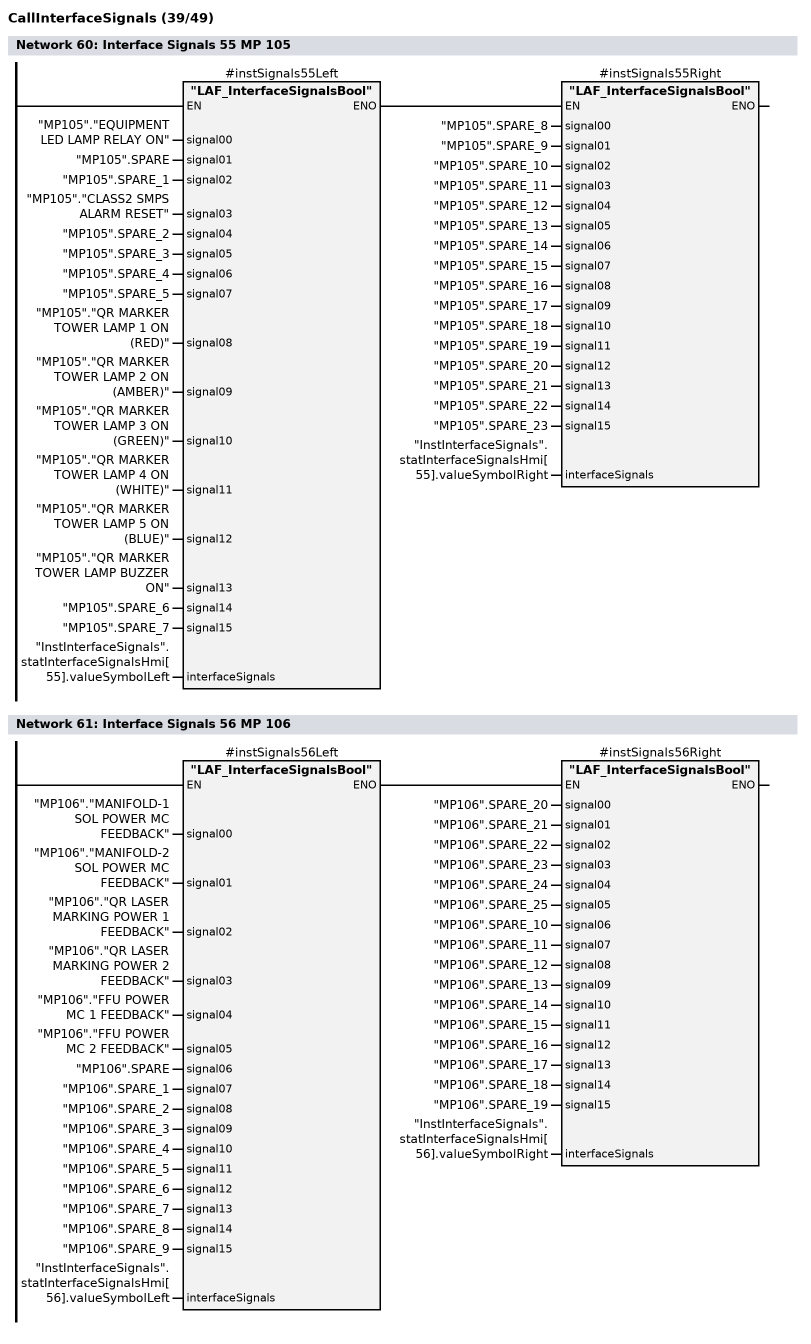
   RUNG wire#powerrail
      #instSignals55Left(signal00 := "MP105"."EQUIPMENT LED LAMP RELAY ON", signal01 := "MP105".SPARE, signal02 := "MP105".SPARE_1, signal03 := "MP105"."CLASS2 SMPS ALARM RESET", signal04 := "MP105".SPARE_2, signal05 := "MP105".SPARE_3, signal06 := "MP105".SPARE_4, signal07 := "MP105".SPARE_5, signal08 := "MP105"."QR MARKER TOWER LAMP 1 ON (RED)", signal09 := "MP105"."QR MARKER TOWER LAMP 2 ON (AMBER)", signal10 := "MP105"."QR MARKER TOWER LAMP 3 ON (GREEN)", signal11 := "MP105"."QR MARKER TOWER LAMP 4 ON (WHITE)", signal12 := "MP105"."QR MARKER TOWER LAMP 5 ON (BLUE)", signal13 := "MP105"."QR MARKER TOWER LAMP BUZZER ON", signal14 := "MP105".SPARE_6, signal15 := "MP105".SPARE_7, interfaceSignals := "InstInterfaceSignals".statInterfaceSignalsHmi[55].valueSymbolLeft)
      #instSignals55Right(signal00 := "MP105".SPARE_8, signal01 := "MP105".SPARE_9, signal02 := "MP105".SPARE_10, signal03 := "MP105".SPARE_11, signal04 := "MP105".SPARE_12, signal05 := "MP105".SPARE_13, signal06 := "MP105".SPARE_14, signal07 := "MP105".SPARE_15, signal08 := "MP105".SPARE_16, signal09 := "MP105".SPARE_17, signal10 := "MP105".SPARE_18, signal11 := "MP105".SPARE_19, signal12 := "MP105".SPARE_20, signal13 := "MP105".SPARE_21, signal14 := "MP105".SPARE_22, signal15 := "MP105".SPARE_23, interfaceSignals := "InstInterfaceSignals".statInterfaceSignalsHmi[55].valueSymbolRight)
   END_RUNG
   // the same network as SCL:
   #instSignals55Left(signal00 := "MP105"."EQUIPMENT LED LAMP RELAY ON",   // "LAF_InterfaceSignalsBool"
                      signal01 := "MP105".SPARE,
                      signal02 := "MP105".SPARE_1,
                      signal03 := "MP105"."CLASS2 SMPS ALARM RESET",
                      signal04 := "MP105".SPARE_2,
                      signal05 := "MP105".SPARE_3,
                      signal06 := "MP105".SPARE_4,
                      signal07 := "MP105".SPARE_5,
                      signal08 := "MP105"."QR MARKER TOWER LAMP 1 ON (RED)",
                      signal09 := "MP105"."QR MARKER TOWER LAMP 2 ON (AMBER)",
                      signal10 := "MP105"."QR MARKER TOWER LAMP 3 ON (GREEN)",
                      signal11 := "MP105"."QR MARKER TOWER LAMP 4 ON (WHITE)",
                      signal12 := "MP105"."QR MARKER TOWER LAMP 5 ON (BLUE)",
                      signal13 := "MP105"."QR MARKER TOWER LAMP BUZZER ON",
                      signal14 := "MP105".SPARE_6,
                      signal15 := "MP105".SPARE_7,
                      interfaceSignals := "InstInterfaceSignals".statInterfaceSignalsHmi[55].valueSymbolLeft,
                      ENO => #_w1);
   IF #_w1 THEN
       #instSignals55Right(signal00 := "MP105".SPARE_8,   // "LAF_InterfaceSignalsBool"
                           signal01 := "MP105".SPARE_9,
                           signal02 := "MP105".SPARE_10,
                           signal03 := "MP105".SPARE_11,
                           signal04 := "MP105".SPARE_12,
                           signal05 := "MP105".SPARE_13,
                           signal06 := "MP105".SPARE_14,
                           signal07 := "MP105".SPARE_15,
                           signal08 := "MP105".SPARE_16,
                           signal09 := "MP105".SPARE_17,
                           signal10 := "MP105".SPARE_18,
                           signal11 := "MP105".SPARE_19,
                           signal12 := "MP105".SPARE_20,
                           signal13 := "MP105".SPARE_21,
                           signal14 := "MP105".SPARE_22,
                           signal15 := "MP105".SPARE_23,
                           interfaceSignals := "InstInterfaceSignals".statInterfaceSignalsHmi[55].valueSymbolRight);
   END_IF;
END_REGION

REGION Network 61: Interface Signals 56 MP 106
   RUNG wire#powerrail
      #instSignals56Left(signal00 := "MP106"."MANIFOLD-1 SOL POWER MC FEEDBACK", signal01 := "MP106"."MANIFOLD-2 SOL POWER MC FEEDBACK", signal02 := "MP106"."QR LASER MARKING POWER 1 FEEDBACK", signal03 := "MP106"."QR LASER MARKING POWER 2 FEEDBACK", signal04 := "MP106"."FFU POWER MC 1 FEEDBACK", signal05 := "MP106"."FFU POWER MC 2 FEEDBACK", signal06 := "MP106".SPARE, signal07 := "MP106".SPARE_1, signal08 := "MP106".SPARE_2, signal09 := "MP106".SPARE_3, signal10 := "MP106".SPARE_4, signal11 := "MP106".SPARE_5, signal12 := "MP106".SPARE_6, signal13 := "MP106".SPARE_7, signal14 := "MP106".SPARE_8, signal15 := "MP106".SPARE_9, interfaceSignals := "InstInterfaceSignals".statInterfaceSignalsHmi[56].valueSymbolLeft)
      #instSignals56Right(signal00 := "MP106".SPARE_20, signal01 := "MP106".SPARE_21, signal02 := "MP106".SPARE_22, signal03 := "MP106".SPARE_23, signal04 := "MP106".SPARE_24, signal05 := "MP106".SPARE_25, signal06 := "MP106".SPARE_10, signal07 := "MP106".SPARE_11, signal08 := "MP106".SPARE_12, signal09 := "MP106".SPARE_13, signal10 := "MP106".SPARE_14, signal11 := "MP106".SPARE_15, signal12 := "MP106".SPARE_16, signal13 := "MP106".SPARE_17, signal14 := "MP106".SPARE_18, signal15 := "MP106".SPARE_19, interfaceSignals := "InstInterfaceSignals".statInterfaceSignalsHmi[56].valueSymbolRight)
   END_RUNG
   // the same network as SCL:
   #instSignals56Left(signal00 := "MP106"."MANIFOLD-1 SOL POWER MC FEEDBACK",   // "LAF_InterfaceSignalsBool"
                      signal01 := "MP106"."MANIFOLD-2 SOL POWER MC FEEDBACK",
                      signal02 := "MP106"."QR LASER MARKING POWER 1 FEEDBACK",
                      signal03 := "MP106"."QR LASER MARKING POWER 2 FEEDBACK",
                      signal04 := "MP106"."FFU POWER MC 1 FEEDBACK",
                      signal05 := "MP106"."FFU POWER MC 2 FEEDBACK",
                      signal06 := "MP106".SPARE,
                      signal07 := "MP106".SPARE_1,
                      signal08 := "MP106".SPARE_2,
                      signal09 := "MP106".SPARE_3,
                      signal10 := "MP106".SPARE_4,
                      signal11 := "MP106".SPARE_5,
                      signal12 := "MP106".SPARE_6,
                      signal13 := "MP106".SPARE_7,
                      signal14 := "MP106".SPARE_8,
                      signal15 := "MP106".SPARE_9,
                      interfaceSignals := "InstInterfaceSignals".statInterfaceSignalsHmi[56].valueSymbolLeft,
                      ENO => #_w1);
   IF #_w1 THEN
       #instSignals56Right(signal00 := "MP106".SPARE_20,   // "LAF_InterfaceSignalsBool"
                           signal01 := "MP106".SPARE_21,
                           signal02 := "MP106".SPARE_22,
                           signal03 := "MP106".SPARE_23,
                           signal04 := "MP106".SPARE_24,
                           signal05 := "MP106".SPARE_25,
                           signal06 := "MP106".SPARE_10,
                           signal07 := "MP106".SPARE_11,
                           signal08 := "MP106".SPARE_12,
                           signal09 := "MP106".SPARE_13,
                           signal10 := "MP106".SPARE_14,
                           signal11 := "MP106".SPARE_15,
                           signal12 := "MP106".SPARE_16,
                           signal13 := "MP106".SPARE_17,
                           signal14 := "MP106".SPARE_18,
                           signal15 := "MP106".SPARE_19,
                           interfaceSignals := "InstInterfaceSignals".statInterfaceSignalsHmi[56].valueSymbolRight);
   END_IF;
END_REGION

REGION Network 62: Interface Signals 57 MP 107
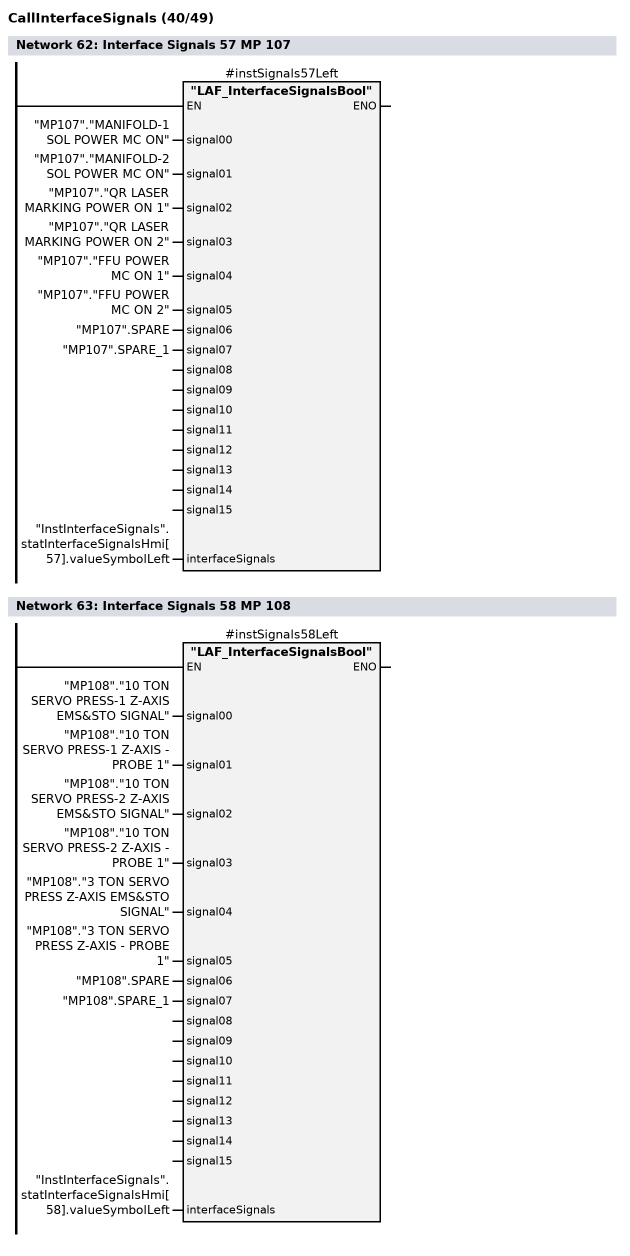
   RUNG wire#powerrail
      #instSignals57Left(signal00 := "MP107"."MANIFOLD-1 SOL POWER MC ON", signal01 := "MP107"."MANIFOLD-2 SOL POWER MC ON", signal02 := "MP107"."QR LASER MARKING POWER ON 1", signal03 := "MP107"."QR LASER MARKING POWER ON 2", signal04 := "MP107"."FFU POWER MC ON 1", signal05 := "MP107"."FFU POWER MC ON 2", signal06 := "MP107".SPARE, signal07 := "MP107".SPARE_1, signal08 :=, signal09 :=, signal10 :=, signal11 :=, signal12 :=, signal13 :=, signal14 :=, signal15 :=, interfaceSignals := "InstInterfaceSignals".statInterfaceSignalsHmi[57].valueSymbolLeft)
   END_RUNG
   // the same network as SCL:
   #instSignals57Left(signal00 := "MP107"."MANIFOLD-1 SOL POWER MC ON",   // "LAF_InterfaceSignalsBool"
                      signal01 := "MP107"."MANIFOLD-2 SOL POWER MC ON",
                      signal02 := "MP107"."QR LASER MARKING POWER ON 1",
                      signal03 := "MP107"."QR LASER MARKING POWER ON 2",
                      signal04 := "MP107"."FFU POWER MC ON 1",
                      signal05 := "MP107"."FFU POWER MC ON 2",
                      signal06 := "MP107".SPARE,
                      signal07 := "MP107".SPARE_1,
                      interfaceSignals := "InstInterfaceSignals".statInterfaceSignalsHmi[57].valueSymbolLeft);
END_REGION

REGION Network 63: Interface Signals 58 MP 108
   RUNG wire#powerrail
      #instSignals58Left(signal00 := "MP108"."10 TON SERVO PRESS-1 Z-AXIS EMS&STO SIGNAL", signal01 := "MP108"."10 TON SERVO PRESS-1 Z-AXIS - PROBE 1", signal02 := "MP108"."10 TON SERVO PRESS-2 Z-AXIS EMS&STO SIGNAL", signal03 := "MP108"."10 TON SERVO PRESS-2 Z-AXIS - PROBE 1", signal04 := "MP108"."3 TON SERVO PRESS Z-AXIS EMS&STO SIGNAL", signal05 := "MP108"."3 TON SERVO PRESS Z-AXIS - PROBE 1", signal06 := "MP108".SPARE, signal07 := "MP108".SPARE_1, signal08 :=, signal09 :=, signal10 :=, signal11 :=, signal12 :=, signal13 :=, signal14 :=, signal15 :=, interfaceSignals := "InstInterfaceSignals".statInterfaceSignalsHmi[58].valueSymbolLeft)
   END_RUNG
   // the same network as SCL:
   #instSignals58Left(signal00 := "MP108"."10 TON SERVO PRESS-1 Z-AXIS EMS&STO SIGNAL",   // "LAF_InterfaceSignalsBool"
                      signal01 := "MP108"."10 TON SERVO PRESS-1 Z-AXIS - PROBE 1",
                      signal02 := "MP108"."10 TON SERVO PRESS-2 Z-AXIS EMS&STO SIGNAL",
                      signal03 := "MP108"."10 TON SERVO PRESS-2 Z-AXIS - PROBE 1",
                      signal04 := "MP108"."3 TON SERVO PRESS Z-AXIS EMS&STO SIGNAL",
                      signal05 := "MP108"."3 TON SERVO PRESS Z-AXIS - PROBE 1",
                      signal06 := "MP108".SPARE,
                      signal07 := "MP108".SPARE_1,
                      interfaceSignals := "InstInterfaceSignals".statInterfaceSignalsHmi[58].valueSymbolLeft);
END_REGION

REGION Network 64: Interface Signals 59 MP 109
END_REGION

REGION Network 65: Interface Signals 60 SP 201
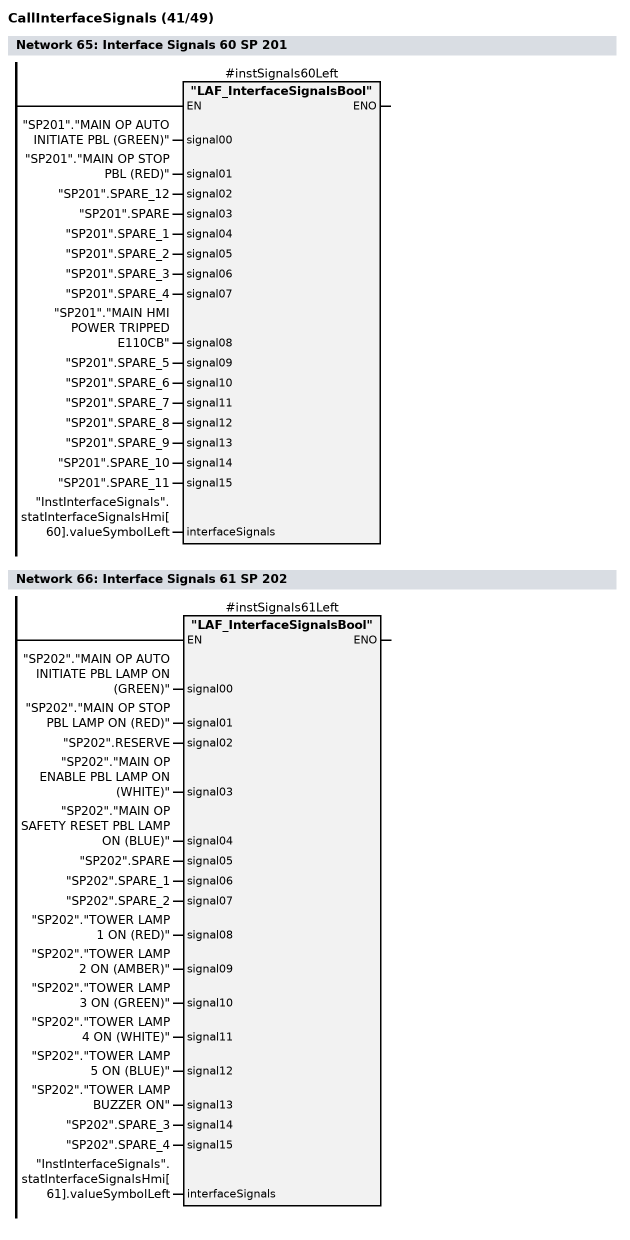
   RUNG wire#powerrail
      #instSignals60Left(signal00 := "SP201"."MAIN OP AUTO INITIATE PBL (GREEN)", signal01 := "SP201"."MAIN OP STOP PBL (RED)", signal02 := "SP201".SPARE_12, signal03 := "SP201".SPARE, signal04 := "SP201".SPARE_1, signal05 := "SP201".SPARE_2, signal06 := "SP201".SPARE_3, signal07 := "SP201".SPARE_4, signal08 := "SP201"."MAIN HMI POWER TRIPPED E110CB", signal09 := "SP201".SPARE_5, signal10 := "SP201".SPARE_6, signal11 := "SP201".SPARE_7, signal12 := "SP201".SPARE_8, signal13 := "SP201".SPARE_9, signal14 := "SP201".SPARE_10, signal15 := "SP201".SPARE_11, interfaceSignals := "InstInterfaceSignals".statInterfaceSignalsHmi[60].valueSymbolLeft)
   END_RUNG
   // the same network as SCL:
   #instSignals60Left(signal00 := "SP201"."MAIN OP AUTO INITIATE PBL (GREEN)",   // "LAF_InterfaceSignalsBool"
                      signal01 := "SP201"."MAIN OP STOP PBL (RED)",
                      signal02 := "SP201".SPARE_12,
                      signal03 := "SP201".SPARE,
                      signal04 := "SP201".SPARE_1,
                      signal05 := "SP201".SPARE_2,
                      signal06 := "SP201".SPARE_3,
                      signal07 := "SP201".SPARE_4,
                      signal08 := "SP201"."MAIN HMI POWER TRIPPED E110CB",
                      signal09 := "SP201".SPARE_5,
                      signal10 := "SP201".SPARE_6,
                      signal11 := "SP201".SPARE_7,
                      signal12 := "SP201".SPARE_8,
                      signal13 := "SP201".SPARE_9,
                      signal14 := "SP201".SPARE_10,
                      signal15 := "SP201".SPARE_11,
                      interfaceSignals := "InstInterfaceSignals".statInterfaceSignalsHmi[60].valueSymbolLeft);
END_REGION

REGION Network 66: Interface Signals 61 SP 202
   RUNG wire#powerrail
      #instSignals61Left(signal00 := "SP202"."MAIN OP AUTO INITIATE PBL LAMP ON (GREEN)", signal01 := "SP202"."MAIN OP STOP PBL LAMP ON (RED)", signal02 := "SP202".RESERVE, signal03 := "SP202"."MAIN OP ENABLE PBL LAMP ON (WHITE)", signal04 := "SP202"."MAIN OP SAFETY RESET PBL LAMP ON (BLUE)", signal05 := "SP202".SPARE, signal06 := "SP202".SPARE_1, signal07 := "SP202".SPARE_2, signal08 := "SP202"."TOWER LAMP 1 ON (RED)", signal09 := "SP202"."TOWER LAMP 2 ON (AMBER)", signal10 := "SP202"."TOWER LAMP 3 ON (GREEN)", signal11 := "SP202"."TOWER LAMP 4 ON (WHITE)", signal12 := "SP202"."TOWER LAMP 5 ON (BLUE)", signal13 := "SP202"."TOWER LAMP BUZZER ON", signal14 := "SP202".SPARE_3, signal15 := "SP202".SPARE_4, interfaceSignals := "InstInterfaceSignals".statInterfaceSignalsHmi[61].valueSymbolLeft)
   END_RUNG
   // the same network as SCL:
   #instSignals61Left(signal00 := "SP202"."MAIN OP AUTO INITIATE PBL LAMP ON (GREEN)",   // "LAF_InterfaceSignalsBool"
                      signal01 := "SP202"."MAIN OP STOP PBL LAMP ON (RED)",
                      signal02 := "SP202".RESERVE,
                      signal03 := "SP202"."MAIN OP ENABLE PBL LAMP ON (WHITE)",
                      signal04 := "SP202"."MAIN OP SAFETY RESET PBL LAMP ON (BLUE)",
                      signal05 := "SP202".SPARE,
                      signal06 := "SP202".SPARE_1,
                      signal07 := "SP202".SPARE_2,
                      signal08 := "SP202"."TOWER LAMP 1 ON (RED)",
                      signal09 := "SP202"."TOWER LAMP 2 ON (AMBER)",
                      signal10 := "SP202"."TOWER LAMP 3 ON (GREEN)",
                      signal11 := "SP202"."TOWER LAMP 4 ON (WHITE)",
                      signal12 := "SP202"."TOWER LAMP 5 ON (BLUE)",
                      signal13 := "SP202"."TOWER LAMP BUZZER ON",
                      signal14 := "SP202".SPARE_3,
                      signal15 := "SP202".SPARE_4,
                      interfaceSignals := "InstInterfaceSignals".statInterfaceSignalsHmi[61].valueSymbolLeft);
END_REGION

REGION Network 67: Interface Signals 62 SP 203
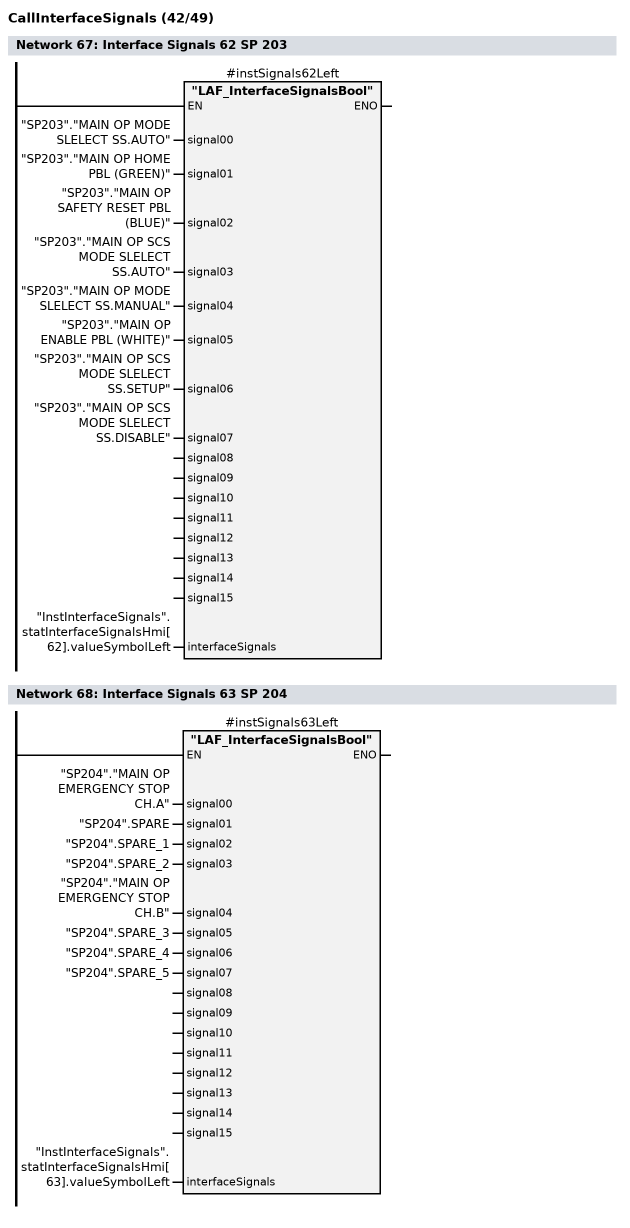
   RUNG wire#powerrail
      #instSignals62Left(signal00 := "SP203"."MAIN OP MODE SLELECT SS.AUTO", signal01 := "SP203"."MAIN OP HOME PBL (GREEN)", signal02 := "SP203"."MAIN OP SAFETY RESET PBL (BLUE)", signal03 := "SP203"."MAIN OP SCS MODE SLELECT SS.AUTO", signal04 := "SP203"."MAIN OP MODE SLELECT SS.MANUAL", signal05 := "SP203"."MAIN OP ENABLE PBL (WHITE)", signal06 := "SP203"."MAIN OP SCS MODE SLELECT SS.SETUP", signal07 := "SP203"."MAIN OP SCS MODE SLELECT SS.DISABLE", signal08 :=, signal09 :=, signal10 :=, signal11 :=, signal12 :=, signal13 :=, signal14 :=, signal15 :=, interfaceSignals := "InstInterfaceSignals".statInterfaceSignalsHmi[62].valueSymbolLeft)
   END_RUNG
   // the same network as SCL:
   #instSignals62Left(signal00 := "SP203"."MAIN OP MODE SLELECT SS.AUTO",   // "LAF_InterfaceSignalsBool"
                      signal01 := "SP203"."MAIN OP HOME PBL (GREEN)",
                      signal02 := "SP203"."MAIN OP SAFETY RESET PBL (BLUE)",
                      signal03 := "SP203"."MAIN OP SCS MODE SLELECT SS.AUTO",
                      signal04 := "SP203"."MAIN OP MODE SLELECT SS.MANUAL",
                      signal05 := "SP203"."MAIN OP ENABLE PBL (WHITE)",
                      signal06 := "SP203"."MAIN OP SCS MODE SLELECT SS.SETUP",
                      signal07 := "SP203"."MAIN OP SCS MODE SLELECT SS.DISABLE",
                      interfaceSignals := "InstInterfaceSignals".statInterfaceSignalsHmi[62].valueSymbolLeft);
END_REGION

REGION Network 68: Interface Signals 63 SP 204
   RUNG wire#powerrail
      #instSignals63Left(signal00 := "SP204"."MAIN OP EMERGENCY STOP CH.A", signal01 := "SP204".SPARE, signal02 := "SP204".SPARE_1, signal03 := "SP204".SPARE_2, signal04 := "SP204"."MAIN OP EMERGENCY STOP CH.B", signal05 := "SP204".SPARE_3, signal06 := "SP204".SPARE_4, signal07 := "SP204".SPARE_5, signal08 :=, signal09 :=, signal10 :=, signal11 :=, signal12 :=, signal13 :=, signal14 :=, signal15 :=, interfaceSignals := "InstInterfaceSignals".statInterfaceSignalsHmi[63].valueSymbolLeft)
   END_RUNG
   // the same network as SCL:
   #instSignals63Left(signal00 := "SP204"."MAIN OP EMERGENCY STOP CH.A",   // "LAF_InterfaceSignalsBool"
                      signal01 := "SP204".SPARE,
                      signal02 := "SP204".SPARE_1,
                      signal03 := "SP204".SPARE_2,
                      signal04 := "SP204"."MAIN OP EMERGENCY STOP CH.B",
                      signal05 := "SP204".SPARE_3,
                      signal06 := "SP204".SPARE_4,
                      signal07 := "SP204".SPARE_5,
                      interfaceSignals := "InstInterfaceSignals".statInterfaceSignalsHmi[63].valueSymbolLeft);
END_REGION

REGION Network 69: Interface Signals 64 SP 205
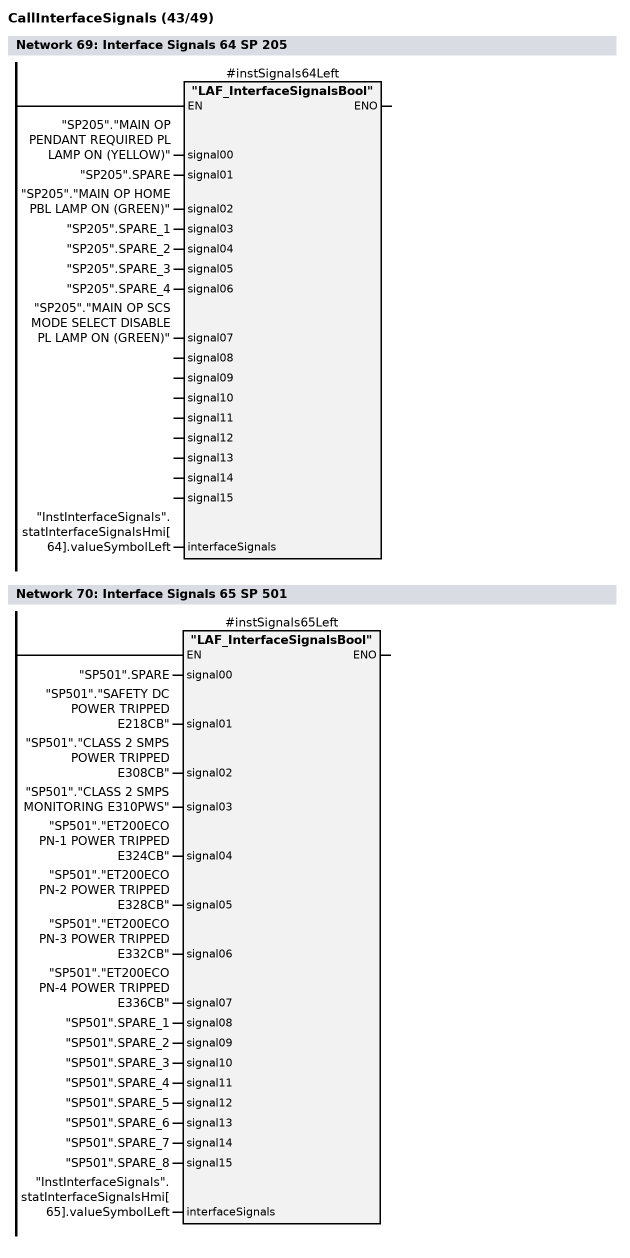
   RUNG wire#powerrail
      #instSignals64Left(signal00 := "SP205"."MAIN OP PENDANT REQUIRED PL LAMP ON (YELLOW)", signal01 := "SP205".SPARE, signal02 := "SP205"."MAIN OP HOME PBL LAMP ON (GREEN)", signal03 := "SP205".SPARE_1, signal04 := "SP205".SPARE_2, signal05 := "SP205".SPARE_3, signal06 := "SP205".SPARE_4, signal07 := "SP205"."MAIN OP SCS MODE SELECT DISABLE PL LAMP ON (GREEN)", signal08 :=, signal09 :=, signal10 :=, signal11 :=, signal12 :=, signal13 :=, signal14 :=, signal15 :=, interfaceSignals := "InstInterfaceSignals".statInterfaceSignalsHmi[64].valueSymbolLeft)
   END_RUNG
   // the same network as SCL:
   #instSignals64Left(signal00 := "SP205"."MAIN OP PENDANT REQUIRED PL LAMP ON (YELLOW)",   // "LAF_InterfaceSignalsBool"
                      signal01 := "SP205".SPARE,
                      signal02 := "SP205"."MAIN OP HOME PBL LAMP ON (GREEN)",
                      signal03 := "SP205".SPARE_1,
                      signal04 := "SP205".SPARE_2,
                      signal05 := "SP205".SPARE_3,
                      signal06 := "SP205".SPARE_4,
                      signal07 := "SP205"."MAIN OP SCS MODE SELECT DISABLE PL LAMP ON (GREEN)",
                      interfaceSignals := "InstInterfaceSignals".statInterfaceSignalsHmi[64].valueSymbolLeft);
END_REGION

REGION Network 70: Interface Signals 65 SP 501
   RUNG wire#powerrail
      #instSignals65Left(signal00 := "SP501".SPARE, signal01 := "SP501"."SAFETY DC POWER TRIPPED E218CB", signal02 := "SP501"."CLASS 2 SMPS POWER TRIPPED E308CB", signal03 := "SP501"."CLASS 2 SMPS MONITORING E310PWS", signal04 := "SP501"."ET200ECO PN-1 POWER TRIPPED E324CB", signal05 := "SP501"."ET200ECO PN-2 POWER TRIPPED E328CB", signal06 := "SP501"."ET200ECO PN-3 POWER TRIPPED E332CB", signal07 := "SP501"."ET200ECO PN-4 POWER TRIPPED E336CB", signal08 := "SP501".SPARE_1, signal09 := "SP501".SPARE_2, signal10 := "SP501".SPARE_3, signal11 := "SP501".SPARE_4, signal12 := "SP501".SPARE_5, signal13 := "SP501".SPARE_6, signal14 := "SP501".SPARE_7, signal15 := "SP501".SPARE_8, interfaceSignals := "InstInterfaceSignals".statInterfaceSignalsHmi[65].valueSymbolLeft)
   END_RUNG
   // the same network as SCL:
   #instSignals65Left(signal00 := "SP501".SPARE,   // "LAF_InterfaceSignalsBool"
                      signal01 := "SP501"."SAFETY DC POWER TRIPPED E218CB",
                      signal02 := "SP501"."CLASS 2 SMPS POWER TRIPPED E308CB",
                      signal03 := "SP501"."CLASS 2 SMPS MONITORING E310PWS",
                      signal04 := "SP501"."ET200ECO PN-1 POWER TRIPPED E324CB",
                      signal05 := "SP501"."ET200ECO PN-2 POWER TRIPPED E328CB",
                      signal06 := "SP501"."ET200ECO PN-3 POWER TRIPPED E332CB",
                      signal07 := "SP501"."ET200ECO PN-4 POWER TRIPPED E336CB",
                      signal08 := "SP501".SPARE_1,
                      signal09 := "SP501".SPARE_2,
                      signal10 := "SP501".SPARE_3,
                      signal11 := "SP501".SPARE_4,
                      signal12 := "SP501".SPARE_5,
                      signal13 := "SP501".SPARE_6,
                      signal14 := "SP501".SPARE_7,
                      signal15 := "SP501".SPARE_8,
                      interfaceSignals := "InstInterfaceSignals".statInterfaceSignalsHmi[65].valueSymbolLeft);
END_REGION

REGION Network 71: Interface Signals 66 SP 502
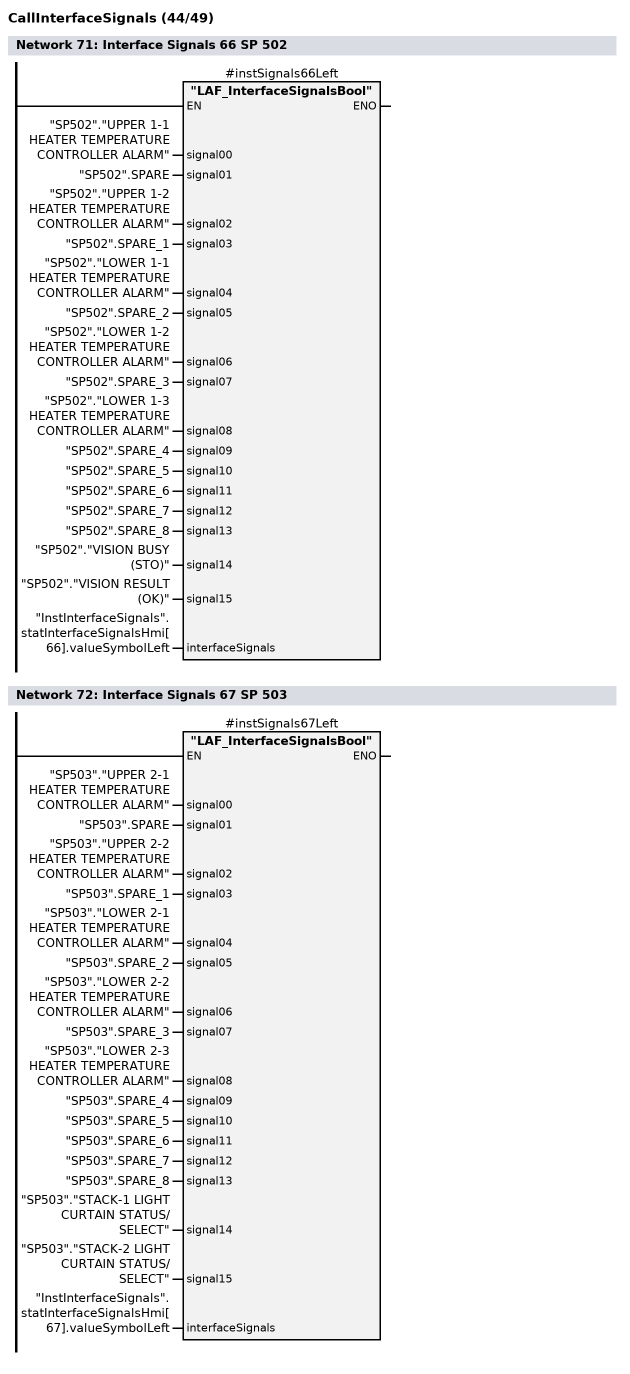
   RUNG wire#powerrail
      #instSignals66Left(signal00 := "SP502"."UPPER 1-1 HEATER TEMPERATURE CONTROLLER ALARM", signal01 := "SP502".SPARE, signal02 := "SP502"."UPPER 1-2 HEATER TEMPERATURE CONTROLLER ALARM", signal03 := "SP502".SPARE_1, signal04 := "SP502"."LOWER 1-1 HEATER TEMPERATURE CONTROLLER ALARM", signal05 := "SP502".SPARE_2, signal06 := "SP502"."LOWER 1-2 HEATER TEMPERATURE CONTROLLER ALARM", signal07 := "SP502".SPARE_3, signal08 := "SP502"."LOWER 1-3 HEATER TEMPERATURE CONTROLLER ALARM", signal09 := "SP502".SPARE_4, signal10 := "SP502".SPARE_5, signal11 := "SP502".SPARE_6, signal12 := "SP502".SPARE_7, signal13 := "SP502".SPARE_8, signal14 := "SP502"."VISION BUSY (STO)", signal15 := "SP502"."VISION RESULT (OK)", interfaceSignals := "InstInterfaceSignals".statInterfaceSignalsHmi[66].valueSymbolLeft)
   END_RUNG
   // the same network as SCL:
   #instSignals66Left(signal00 := "SP502"."UPPER 1-1 HEATER TEMPERATURE CONTROLLER ALARM",   // "LAF_InterfaceSignalsBool"
                      signal01 := "SP502".SPARE,
                      signal02 := "SP502"."UPPER 1-2 HEATER TEMPERATURE CONTROLLER ALARM",
                      signal03 := "SP502".SPARE_1,
                      signal04 := "SP502"."LOWER 1-1 HEATER TEMPERATURE CONTROLLER ALARM",
                      signal05 := "SP502".SPARE_2,
                      signal06 := "SP502"."LOWER 1-2 HEATER TEMPERATURE CONTROLLER ALARM",
                      signal07 := "SP502".SPARE_3,
                      signal08 := "SP502"."LOWER 1-3 HEATER TEMPERATURE CONTROLLER ALARM",
                      signal09 := "SP502".SPARE_4,
                      signal10 := "SP502".SPARE_5,
                      signal11 := "SP502".SPARE_6,
                      signal12 := "SP502".SPARE_7,
                      signal13 := "SP502".SPARE_8,
                      signal14 := "SP502"."VISION BUSY (STO)",
                      signal15 := "SP502"."VISION RESULT (OK)",
                      interfaceSignals := "InstInterfaceSignals".statInterfaceSignalsHmi[66].valueSymbolLeft);
END_REGION

REGION Network 72: Interface Signals 67 SP 503
   RUNG wire#powerrail
      #instSignals67Left(signal00 := "SP503"."UPPER 2-1 HEATER TEMPERATURE CONTROLLER ALARM", signal01 := "SP503".SPARE, signal02 := "SP503"."UPPER 2-2 HEATER TEMPERATURE CONTROLLER ALARM", signal03 := "SP503".SPARE_1, signal04 := "SP503"."LOWER 2-1 HEATER TEMPERATURE CONTROLLER ALARM", signal05 := "SP503".SPARE_2, signal06 := "SP503"."LOWER 2-2 HEATER TEMPERATURE CONTROLLER ALARM", signal07 := "SP503".SPARE_3, signal08 := "SP503"."LOWER 2-3 HEATER TEMPERATURE CONTROLLER ALARM", signal09 := "SP503".SPARE_4, signal10 := "SP503".SPARE_5, signal11 := "SP503".SPARE_6, signal12 := "SP503".SPARE_7, signal13 := "SP503".SPARE_8, signal14 := "SP503"."STACK-1 LIGHT CURTAIN STATUS/SELECT", signal15 := "SP503"."STACK-2 LIGHT CURTAIN STATUS/SELECT", interfaceSignals := "InstInterfaceSignals".statInterfaceSignalsHmi[67].valueSymbolLeft)
   END_RUNG
   // the same network as SCL:
   #instSignals67Left(signal00 := "SP503"."UPPER 2-1 HEATER TEMPERATURE CONTROLLER ALARM",   // "LAF_InterfaceSignalsBool"
                      signal01 := "SP503".SPARE,
                      signal02 := "SP503"."UPPER 2-2 HEATER TEMPERATURE CONTROLLER ALARM",
                      signal03 := "SP503".SPARE_1,
                      signal04 := "SP503"."LOWER 2-1 HEATER TEMPERATURE CONTROLLER ALARM",
                      signal05 := "SP503".SPARE_2,
                      signal06 := "SP503"."LOWER 2-2 HEATER TEMPERATURE CONTROLLER ALARM",
                      signal07 := "SP503".SPARE_3,
                      signal08 := "SP503"."LOWER 2-3 HEATER TEMPERATURE CONTROLLER ALARM",
                      signal09 := "SP503".SPARE_4,
                      signal10 := "SP503".SPARE_5,
                      signal11 := "SP503".SPARE_6,
                      signal12 := "SP503".SPARE_7,
                      signal13 := "SP503".SPARE_8,
                      signal14 := "SP503"."STACK-1 LIGHT CURTAIN STATUS/SELECT",
                      signal15 := "SP503"."STACK-2 LIGHT CURTAIN STATUS/SELECT",
                      interfaceSignals := "InstInterfaceSignals".statInterfaceSignalsHmi[67].valueSymbolLeft);
END_REGION

REGION Network 73: Interface Signals 68 SP 504
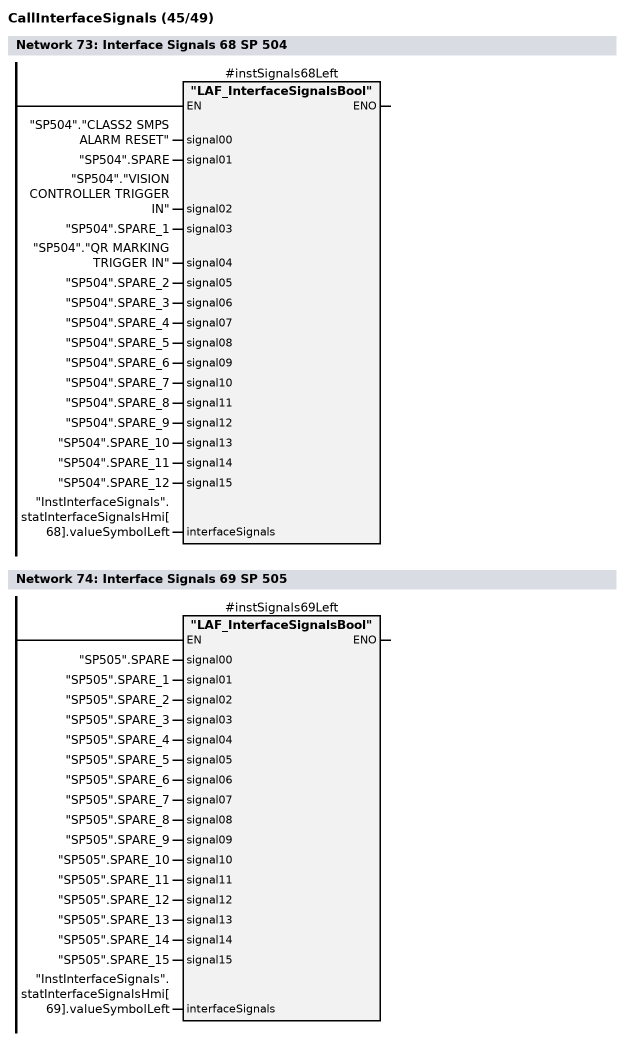
   RUNG wire#powerrail
      #instSignals68Left(signal00 := "SP504"."CLASS2 SMPS ALARM RESET", signal01 := "SP504".SPARE, signal02 := "SP504"."VISION CONTROLLER TRIGGER IN", signal03 := "SP504".SPARE_1, signal04 := "SP504"."QR MARKING TRIGGER IN", signal05 := "SP504".SPARE_2, signal06 := "SP504".SPARE_3, signal07 := "SP504".SPARE_4, signal08 := "SP504".SPARE_5, signal09 := "SP504".SPARE_6, signal10 := "SP504".SPARE_7, signal11 := "SP504".SPARE_8, signal12 := "SP504".SPARE_9, signal13 := "SP504".SPARE_10, signal14 := "SP504".SPARE_11, signal15 := "SP504".SPARE_12, interfaceSignals := "InstInterfaceSignals".statInterfaceSignalsHmi[68].valueSymbolLeft)
   END_RUNG
   // the same network as SCL:
   #instSignals68Left(signal00 := "SP504"."CLASS2 SMPS ALARM RESET",   // "LAF_InterfaceSignalsBool"
                      signal01 := "SP504".SPARE,
                      signal02 := "SP504"."VISION CONTROLLER TRIGGER IN",
                      signal03 := "SP504".SPARE_1,
                      signal04 := "SP504"."QR MARKING TRIGGER IN",
                      signal05 := "SP504".SPARE_2,
                      signal06 := "SP504".SPARE_3,
                      signal07 := "SP504".SPARE_4,
                      signal08 := "SP504".SPARE_5,
                      signal09 := "SP504".SPARE_6,
                      signal10 := "SP504".SPARE_7,
                      signal11 := "SP504".SPARE_8,
                      signal12 := "SP504".SPARE_9,
                      signal13 := "SP504".SPARE_10,
                      signal14 := "SP504".SPARE_11,
                      signal15 := "SP504".SPARE_12,
                      interfaceSignals := "InstInterfaceSignals".statInterfaceSignalsHmi[68].valueSymbolLeft);
END_REGION

REGION Network 74: Interface Signals 69 SP 505
   RUNG wire#powerrail
      #instSignals69Left(signal00 := "SP505".SPARE, signal01 := "SP505".SPARE_1, signal02 := "SP505".SPARE_2, signal03 := "SP505".SPARE_3, signal04 := "SP505".SPARE_4, signal05 := "SP505".SPARE_5, signal06 := "SP505".SPARE_6, signal07 := "SP505".SPARE_7, signal08 := "SP505".SPARE_8, signal09 := "SP505".SPARE_9, signal10 := "SP505".SPARE_10, signal11 := "SP505".SPARE_11, signal12 := "SP505".SPARE_12, signal13 := "SP505".SPARE_13, signal14 := "SP505".SPARE_14, signal15 := "SP505".SPARE_15, interfaceSignals := "InstInterfaceSignals".statInterfaceSignalsHmi[69].valueSymbolLeft)
   END_RUNG
   // the same network as SCL:
   #instSignals69Left(signal00 := "SP505".SPARE,   // "LAF_InterfaceSignalsBool"
                      signal01 := "SP505".SPARE_1,
                      signal02 := "SP505".SPARE_2,
                      signal03 := "SP505".SPARE_3,
                      signal04 := "SP505".SPARE_4,
                      signal05 := "SP505".SPARE_5,
                      signal06 := "SP505".SPARE_6,
                      signal07 := "SP505".SPARE_7,
                      signal08 := "SP505".SPARE_8,
                      signal09 := "SP505".SPARE_9,
                      signal10 := "SP505".SPARE_10,
                      signal11 := "SP505".SPARE_11,
                      signal12 := "SP505".SPARE_12,
                      signal13 := "SP505".SPARE_13,
                      signal14 := "SP505".SPARE_14,
                      signal15 := "SP505".SPARE_15,
                      interfaceSignals := "InstInterfaceSignals".statInterfaceSignalsHmi[69].valueSymbolLeft);
END_REGION

REGION Network 75: Interface Signals 70 SP 506
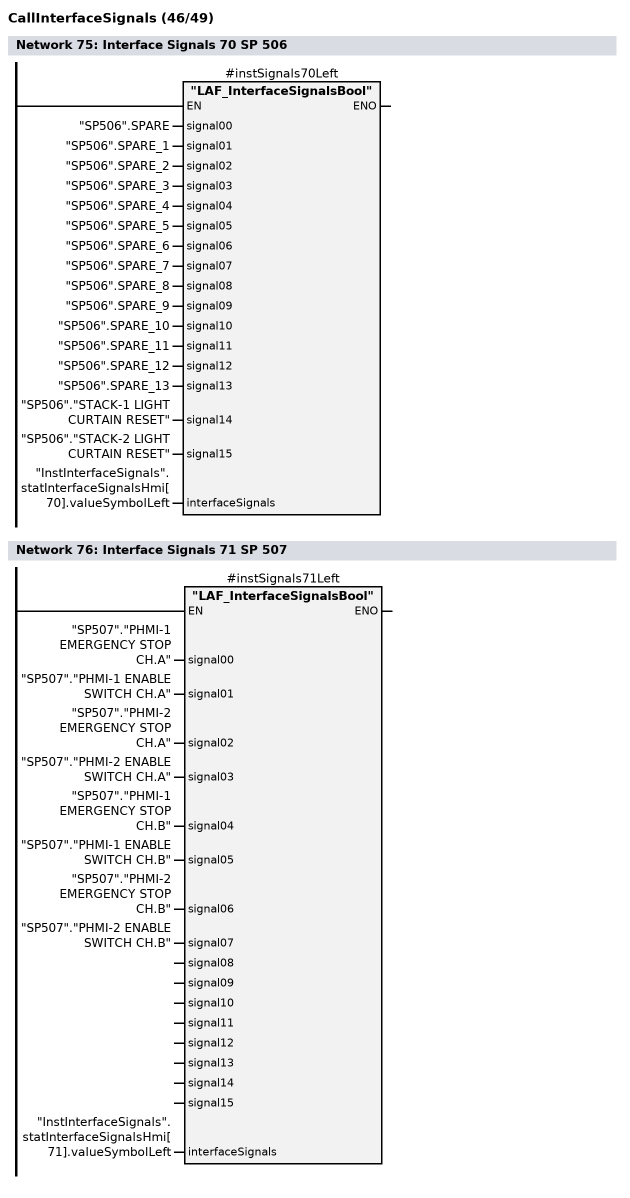
   RUNG wire#powerrail
      #instSignals70Left(signal00 := "SP506".SPARE, signal01 := "SP506".SPARE_1, signal02 := "SP506".SPARE_2, signal03 := "SP506".SPARE_3, signal04 := "SP506".SPARE_4, signal05 := "SP506".SPARE_5, signal06 := "SP506".SPARE_6, signal07 := "SP506".SPARE_7, signal08 := "SP506".SPARE_8, signal09 := "SP506".SPARE_9, signal10 := "SP506".SPARE_10, signal11 := "SP506".SPARE_11, signal12 := "SP506".SPARE_12, signal13 := "SP506".SPARE_13, signal14 := "SP506"."STACK-1 LIGHT CURTAIN RESET", signal15 := "SP506"."STACK-2 LIGHT CURTAIN RESET", interfaceSignals := "InstInterfaceSignals".statInterfaceSignalsHmi[70].valueSymbolLeft)
   END_RUNG
   // the same network as SCL:
   #instSignals70Left(signal00 := "SP506".SPARE,   // "LAF_InterfaceSignalsBool"
                      signal01 := "SP506".SPARE_1,
                      signal02 := "SP506".SPARE_2,
                      signal03 := "SP506".SPARE_3,
                      signal04 := "SP506".SPARE_4,
                      signal05 := "SP506".SPARE_5,
                      signal06 := "SP506".SPARE_6,
                      signal07 := "SP506".SPARE_7,
                      signal08 := "SP506".SPARE_8,
                      signal09 := "SP506".SPARE_9,
                      signal10 := "SP506".SPARE_10,
                      signal11 := "SP506".SPARE_11,
                      signal12 := "SP506".SPARE_12,
                      signal13 := "SP506".SPARE_13,
                      signal14 := "SP506"."STACK-1 LIGHT CURTAIN RESET",
                      signal15 := "SP506"."STACK-2 LIGHT CURTAIN RESET",
                      interfaceSignals := "InstInterfaceSignals".statInterfaceSignalsHmi[70].valueSymbolLeft);
END_REGION

REGION Network 76: Interface Signals 71 SP 507
   RUNG wire#powerrail
      #instSignals71Left(signal00 := "SP507"."PHMI-1 EMERGENCY STOP CH.A", signal01 := "SP507"."PHMI-1 ENABLE SWITCH CH.A", signal02 := "SP507"."PHMI-2 EMERGENCY STOP CH.A", signal03 := "SP507"."PHMI-2 ENABLE SWITCH CH.A", signal04 := "SP507"."PHMI-1 EMERGENCY STOP CH.B", signal05 := "SP507"."PHMI-1 ENABLE SWITCH CH.B", signal06 := "SP507"."PHMI-2 EMERGENCY STOP CH.B", signal07 := "SP507"."PHMI-2 ENABLE SWITCH CH.B", signal08 :=, signal09 :=, signal10 :=, signal11 :=, signal12 :=, signal13 :=, signal14 :=, signal15 :=, interfaceSignals := "InstInterfaceSignals".statInterfaceSignalsHmi[71].valueSymbolLeft)
   END_RUNG
   // the same network as SCL:
   #instSignals71Left(signal00 := "SP507"."PHMI-1 EMERGENCY STOP CH.A",   // "LAF_InterfaceSignalsBool"
                      signal01 := "SP507"."PHMI-1 ENABLE SWITCH CH.A",
                      signal02 := "SP507"."PHMI-2 EMERGENCY STOP CH.A",
                      signal03 := "SP507"."PHMI-2 ENABLE SWITCH CH.A",
                      signal04 := "SP507"."PHMI-1 EMERGENCY STOP CH.B",
                      signal05 := "SP507"."PHMI-1 ENABLE SWITCH CH.B",
                      signal06 := "SP507"."PHMI-2 EMERGENCY STOP CH.B",
                      signal07 := "SP507"."PHMI-2 ENABLE SWITCH CH.B",
                      interfaceSignals := "InstInterfaceSignals".statInterfaceSignalsHmi[71].valueSymbolLeft);
END_REGION

REGION Network 77: Interface Signals 72 SP 508
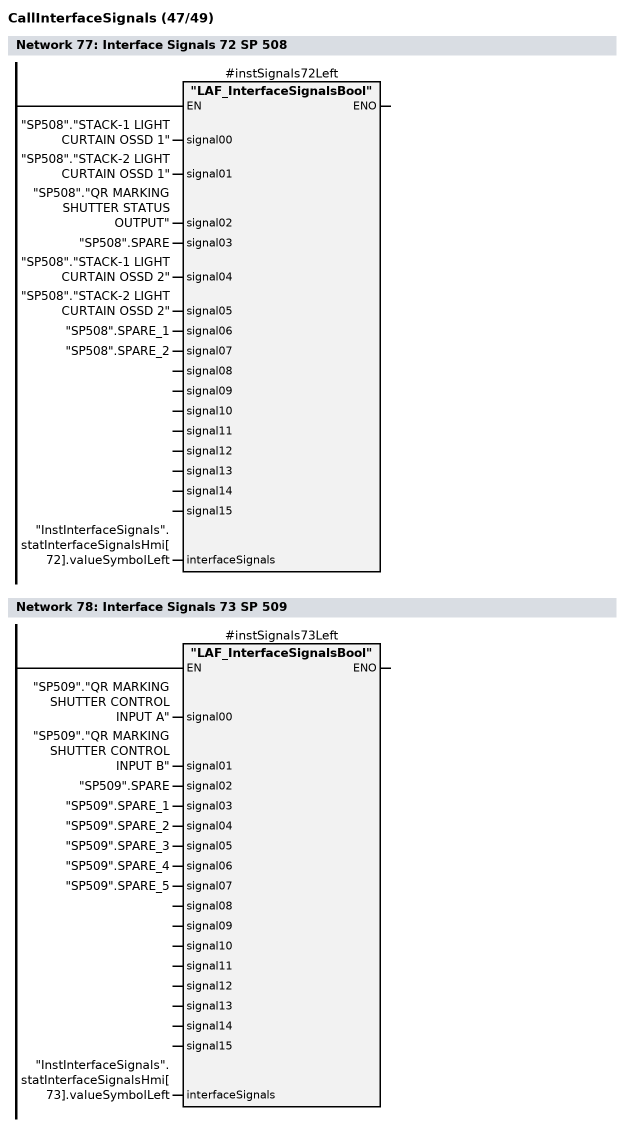
   RUNG wire#powerrail
      #instSignals72Left(signal00 := "SP508"."STACK-1 LIGHT CURTAIN OSSD 1", signal01 := "SP508"."STACK-2 LIGHT CURTAIN OSSD 1", signal02 := "SP508"."QR MARKING SHUTTER STATUS OUTPUT", signal03 := "SP508".SPARE, signal04 := "SP508"."STACK-1 LIGHT CURTAIN OSSD 2", signal05 := "SP508"."STACK-2 LIGHT CURTAIN OSSD 2", signal06 := "SP508".SPARE_1, signal07 := "SP508".SPARE_2, signal08 :=, signal09 :=, signal10 :=, signal11 :=, signal12 :=, signal13 :=, signal14 :=, signal15 :=, interfaceSignals := "InstInterfaceSignals".statInterfaceSignalsHmi[72].valueSymbolLeft)
   END_RUNG
   // the same network as SCL:
   #instSignals72Left(signal00 := "SP508"."STACK-1 LIGHT CURTAIN OSSD 1",   // "LAF_InterfaceSignalsBool"
                      signal01 := "SP508"."STACK-2 LIGHT CURTAIN OSSD 1",
                      signal02 := "SP508"."QR MARKING SHUTTER STATUS OUTPUT",
                      signal03 := "SP508".SPARE,
                      signal04 := "SP508"."STACK-1 LIGHT CURTAIN OSSD 2",
                      signal05 := "SP508"."STACK-2 LIGHT CURTAIN OSSD 2",
                      signal06 := "SP508".SPARE_1,
                      signal07 := "SP508".SPARE_2,
                      interfaceSignals := "InstInterfaceSignals".statInterfaceSignalsHmi[72].valueSymbolLeft);
END_REGION

REGION Network 78: Interface Signals 73 SP 509
   RUNG wire#powerrail
      #instSignals73Left(signal00 := "SP509"."QR MARKING SHUTTER CONTROL INPUT A", signal01 := "SP509"."QR MARKING SHUTTER CONTROL INPUT B", signal02 := "SP509".SPARE, signal03 := "SP509".SPARE_1, signal04 := "SP509".SPARE_2, signal05 := "SP509".SPARE_3, signal06 := "SP509".SPARE_4, signal07 := "SP509".SPARE_5, signal08 :=, signal09 :=, signal10 :=, signal11 :=, signal12 :=, signal13 :=, signal14 :=, signal15 :=, interfaceSignals := "InstInterfaceSignals".statInterfaceSignalsHmi[73].valueSymbolLeft)
   END_RUNG
   // the same network as SCL:
   #instSignals73Left(signal00 := "SP509"."QR MARKING SHUTTER CONTROL INPUT A",   // "LAF_InterfaceSignalsBool"
                      signal01 := "SP509"."QR MARKING SHUTTER CONTROL INPUT B",
                      signal02 := "SP509".SPARE,
                      signal03 := "SP509".SPARE_1,
                      signal04 := "SP509".SPARE_2,
                      signal05 := "SP509".SPARE_3,
                      signal06 := "SP509".SPARE_4,
                      signal07 := "SP509".SPARE_5,
                      interfaceSignals := "InstInterfaceSignals".statInterfaceSignalsHmi[73].valueSymbolLeft);
END_REGION

REGION Network 79: Interface Signals 74 SP 510
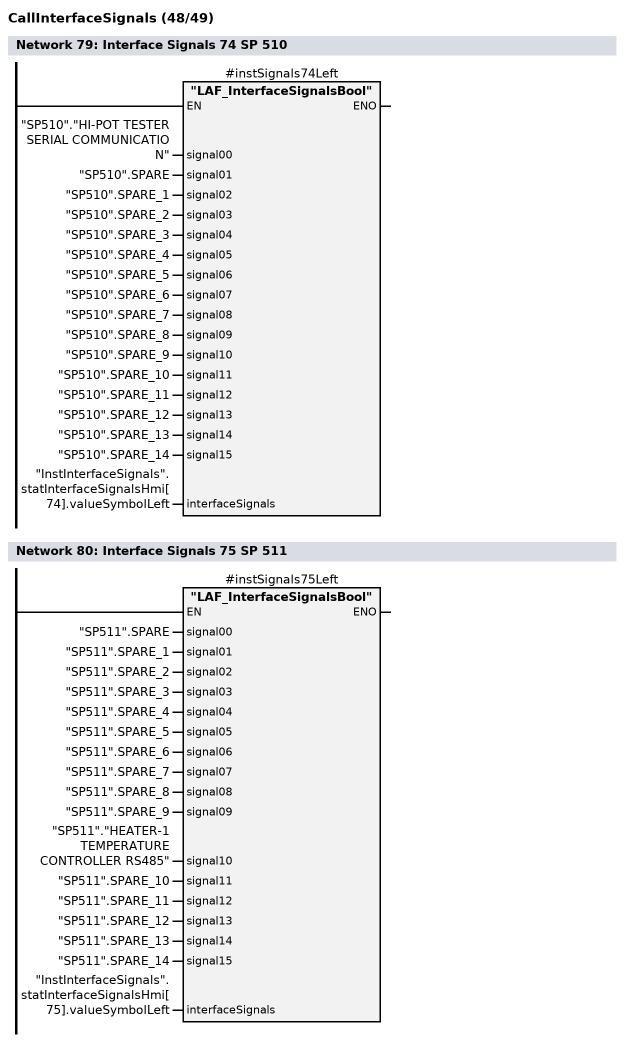
   RUNG wire#powerrail
      #instSignals74Left(signal00 := "SP510"."HI-POT TESTER SERIAL COMMUNICATION", signal01 := "SP510".SPARE, signal02 := "SP510".SPARE_1, signal03 := "SP510".SPARE_2, signal04 := "SP510".SPARE_3, signal05 := "SP510".SPARE_4, signal06 := "SP510".SPARE_5, signal07 := "SP510".SPARE_6, signal08 := "SP510".SPARE_7, signal09 := "SP510".SPARE_8, signal10 := "SP510".SPARE_9, signal11 := "SP510".SPARE_10, signal12 := "SP510".SPARE_11, signal13 := "SP510".SPARE_12, signal14 := "SP510".SPARE_13, signal15 := "SP510".SPARE_14, interfaceSignals := "InstInterfaceSignals".statInterfaceSignalsHmi[74].valueSymbolLeft)
   END_RUNG
   // the same network as SCL:
   #instSignals74Left(signal00 := "SP510"."HI-POT TESTER SERIAL COMMUNICATION",   // "LAF_InterfaceSignalsBool"
                      signal01 := "SP510".SPARE,
                      signal02 := "SP510".SPARE_1,
                      signal03 := "SP510".SPARE_2,
                      signal04 := "SP510".SPARE_3,
                      signal05 := "SP510".SPARE_4,
                      signal06 := "SP510".SPARE_5,
                      signal07 := "SP510".SPARE_6,
                      signal08 := "SP510".SPARE_7,
                      signal09 := "SP510".SPARE_8,
                      signal10 := "SP510".SPARE_9,
                      signal11 := "SP510".SPARE_10,
                      signal12 := "SP510".SPARE_11,
                      signal13 := "SP510".SPARE_12,
                      signal14 := "SP510".SPARE_13,
                      signal15 := "SP510".SPARE_14,
                      interfaceSignals := "InstInterfaceSignals".statInterfaceSignalsHmi[74].valueSymbolLeft);
END_REGION

REGION Network 80: Interface Signals 75 SP 511
   RUNG wire#powerrail
      #instSignals75Left(signal00 := "SP511".SPARE, signal01 := "SP511".SPARE_1, signal02 := "SP511".SPARE_2, signal03 := "SP511".SPARE_3, signal04 := "SP511".SPARE_4, signal05 := "SP511".SPARE_5, signal06 := "SP511".SPARE_6, signal07 := "SP511".SPARE_7, signal08 := "SP511".SPARE_8, signal09 := "SP511".SPARE_9, signal10 := "SP511"."HEATER-1 TEMPERATURE CONTROLLER RS485", signal11 := "SP511".SPARE_10, signal12 := "SP511".SPARE_11, signal13 := "SP511".SPARE_12, signal14 := "SP511".SPARE_13, signal15 := "SP511".SPARE_14, interfaceSignals := "InstInterfaceSignals".statInterfaceSignalsHmi[75].valueSymbolLeft)
   END_RUNG
   // the same network as SCL:
   #instSignals75Left(signal00 := "SP511".SPARE,   // "LAF_InterfaceSignalsBool"
                      signal01 := "SP511".SPARE_1,
                      signal02 := "SP511".SPARE_2,
                      signal03 := "SP511".SPARE_3,
                      signal04 := "SP511".SPARE_4,
                      signal05 := "SP511".SPARE_5,
                      signal06 := "SP511".SPARE_6,
                      signal07 := "SP511".SPARE_7,
                      signal08 := "SP511".SPARE_8,
                      signal09 := "SP511".SPARE_9,
                      signal10 := "SP511"."HEATER-1 TEMPERATURE CONTROLLER RS485",
                      signal11 := "SP511".SPARE_10,
                      signal12 := "SP511".SPARE_11,
                      signal13 := "SP511".SPARE_12,
                      signal14 := "SP511".SPARE_13,
                      signal15 := "SP511".SPARE_14,
                      interfaceSignals := "InstInterfaceSignals".statInterfaceSignalsHmi[75].valueSymbolLeft);
END_REGION

REGION Network 81: Interface Signals 76 SP 512
